KUKA KRL program: MyProgram_047().src

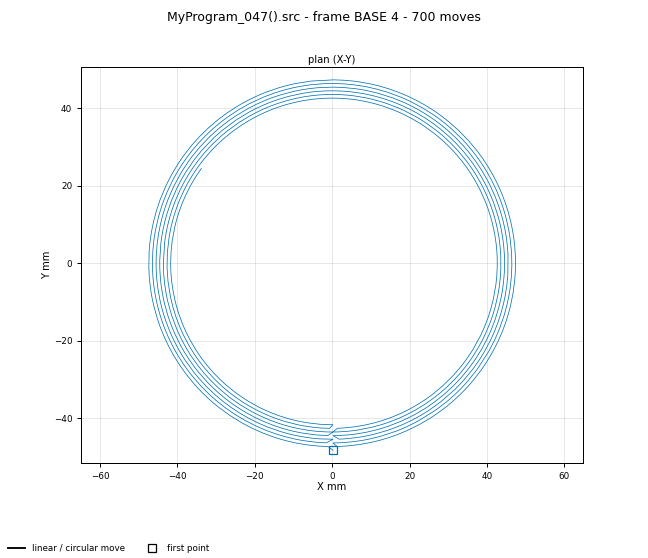
[picture p0: tool path of MyProgram_047().src in frame BASE 4, 700 of 700 moves have a stored position in this frame; points joined in program order, loops and branches not executed]
&ACCESS RVP
&REL 1
&PARAM TEMPLATE = C:\KRC\Roboter\Template\vorgabe
&PARAM EDITMASK = *
DEF MyProgram_047()
; ---- Setting reference (Base) ----
$BASE = BASE_DATA[4]

; --------------------------
; ---- Setting tool (TCP) ----
$TOOL = TOOL_DATA[3]
; --------------------------

$VEL.CP = VEL_APROX_PRINT
Startdeposition()
$VEL.CP = VEL_PRINT
LIN {X 0.2248,Y -48.3264,Z 65,A -97.1945,B 24.8798,C -2.5309,E1 24.997,E2 -179.1657} C_DIS
Enddeposition()
LIN {X 0.2248,Y -48.3264,Z 65,A -97.1945,B 24.8798,C -2.5309,E1 24.997,E2 -179.1657} C_DIS
Startdeposition()
$VEL.CP = VEL_PRINT
LIN {X -1.0477,Y -47.3732,Z 65,A -98.6326,B 24.878,C -2.5491,E1 24.9931,E2 -177.7706} C_DIS
LIN {X -3.5749,Y -47.2498,Z 65,A -101.1612,B 24.8772,C -2.5575,E1 24.9861,E2 -175.2611} C_DIS
LIN {X -6.5546,Y -46.929,Z 65,A -105.0891,B 24.8776,C -2.5533,E1 24.9752,E2 -171.3204} C_DIS
LIN {X -9.2778,Y -46.468,Z 65,A -107.7216,B 24.8764,C -2.5655,E1 24.968,E2 -168.7143} C_DIS
LIN {X -11.575,Y -45.9489,Z 65,A -110.7748,B 24.8766,C -2.5637,E1 24.9597,E2 -165.6528} C_DIS
LIN {X -13.521,Y -45.4144,Z 65,A -113.2414,B 24.8766,C -2.5649,E1 24.9531,E2 -163.1849} C_DIS
LIN {X -15.4389,Y -44.7995,Z 65,A -115.7196,B 24.8764,C -2.5661,E1 24.9465,E2 -160.7051} C_DIS
LIN {X -17.756,Y -43.932,Z 65,A -119.0552,B 24.8766,C -2.5637,E1 24.9378,E2 -157.3566} C_DIS
LIN {X -20.3496,Y -42.7927,Z 65,A -122.8119,B 24.8767,C -2.5626,E1 24.9282,E2 -153.588} C_DIS
LIN {X -23.3064,Y -41.2571,Z 65,A -126.6828,B 24.876,C -2.5702,E1 24.9188,E2 -149.7241} C_DIS
LIN {X -26.4858,Y -39.2912,Z 65,A -131.3289,B 24.8755,C -2.5752,E1 24.9079,E2 -145.0751} C_DIS
LIN {X -29.4186,Y -37.1461,Z 65,A -135.0423,B 24.8738,C -2.5924,E1 24.8996,E2 -141.3894} C_DIS
LIN {X -30.8579,Y -35.9594,Z 65,A -137.3147,B 24.8734,C -2.5964,E1 24.8948,E2 -139.1176} C_DIS
LIN {X -32.1607,Y -34.7995,Z 65,A -139.563,B 24.8732,C -2.5985,E1 24.8901,E2 -136.8654} C_DIS
LIN {X -33.7294,Y -33.2807,Z 65,A -142.3681,B 24.8729,C -2.6017,E1 24.8846,E2 -134.056} C_DIS
LIN {X -35.5399,Y -31.34,Z 65,A -146.1751,B 24.873,C -2.6005,E1 24.8774,E2 -130.2292} C_DIS
LIN {X -37.5818,Y -28.8599,Z 65,A -149.5808,B 24.8715,C -2.616,E1 24.8716,E2 -126.8446} C_DIS
LIN {X -39.2128,Y -26.6015,Z 65,A -153.0058,B 24.8708,C -2.6235,E1 24.8661,E2 -123.4206} C_DIS
LIN {X -40.9588,Y -23.8267,Z 65,A -156.7428,B 24.8695,C -2.6367,E1 24.8607,E2 -119.696} C_DIS
LIN {X -42.1995,Y -21.5519,Z 65,A -160.1247,B 24.869,C -2.6418,E1 24.8563,E2 -116.3083} C_DIS
LIN {X -43.292,Y -19.2649,Z 65,A -163.5194,B 24.8685,C -2.646,E1 24.8523,E2 -112.905} C_DIS
LIN {X -44.419,Y -16.5014,Z 65,A -166.5245,B 24.8667,C -2.6641,E1 24.8493,E2 -109.9264} C_DIS
LIN {X -45.1483,Y -14.3836,Z 65,A -169.6546,B 24.8665,C -2.6665,E1 24.8466,E2 -106.7842} C_DIS
LIN {X -46.0448,Y -11.1877,Z 65,A -173.5161,B 24.8651,C -2.6804,E1 24.8438,E2 -102.9335} C_DIS
LIN {X -46.5143,Y -9.0394,Z 65,A -175.9159,B 24.8639,C -2.6918,E1 24.8425,E2 -100.5468} C_DIS
LIN {X -46.7881,Y -7.4983,Z 65,A -177.7088,B 24.8632,C -2.6989,E1 24.8416,E2 -98.7601} C_DIS
LIN {X -47.0559,Y -5.5702,Z 65,A 179.5109,B 24.863,C -2.7007,E1 24.8406,E2 -95.9675} C_DIS
LIN {X -47.2538,Y -3.5244,Z 65,A 177.0172,B 24.8622,C -2.7083,E1 24.8401,E2 -93.477} C_DIS
LIN {X -47.3725,Y -1.0864,Z 65,A 173.6451,B 24.8618,C -2.7122,E1 24.8398,E2 -90.094} C_DIS
LIN {X -47.2852,Y 3.0683,Z 65,A 169.3289,B 24.8593,C -2.737,E1 24.8402,E2 -85.8111} C_DIS
LIN {X -47.1535,Y 4.676,Z 65,A 167.3632,B 24.8587,C -2.743,E1 24.8407,E2 -83.8478} C_DIS
LIN {X -46.9842,Y 6.1456,Z 65,A 165.4093,B 24.8583,C -2.7465,E1 24.8414,E2 -81.8907} C_DIS
LIN {X -46.6648,Y 8.2283,Z 65,A 162.772,B 24.8576,C -2.7533,E1 24.8426,E2 -79.254} C_DIS
LIN {X -46.1094,Y 10.9184,Z 65,A 159.2452,B 24.8568,C -2.761,E1 24.8447,E2 -75.725} C_DIS
LIN {X -45.3809,Y 13.634,Z 65,A 155.7906,B 24.8558,C -2.7708,E1 24.8473,E2 -72.2736} C_DIS
LIN {X -44.4848,Y 16.3215,Z 65,A 152.1165,B 24.855,C -2.778,E1 24.8507,E2 -68.596} C_DIS
LIN {X -42.9085,Y 20.1037,Z 65,A 148.0403,B 24.8523,C -2.8039,E1 24.8552,E2 -64.5593} C_DIS
LIN {X -41.5375,Y 22.8004,Z 65,A 143.2509,B 24.8527,C -2.7999,E1 24.8615,E2 -59.7346} C_DIS
LIN {X -39.7956,Y 25.7219,Z 65,A 139.6863,B 24.8508,C -2.8183,E1 24.8667,E2 -56.196} C_DIS
LIN {X -38.3081,Y 27.8889,Z 65,A 136.4395,B 24.85,C -2.8259,E1 24.8719,E2 -52.9515} C_DIS
LIN {X -36.3484,Y 30.399,Z 65,A 132.1204,B 24.8496,C -2.8296,E1 24.8795,E2 -48.6212} C_DIS
LIN {X -34.1939,Y 32.8036,Z 65,A 128.7989,B 24.8477,C -2.8469,E1 24.8858,E2 -45.3263} C_DIS
LIN {X -31.929,Y 35.0116,Z 65,A 124.5127,B 24.8475,C -2.8495,E1 24.8945,E2 -41.0286} C_DIS
LIN {X -29.3388,Y 37.2091,Z 65,A 120.4495,B 24.8464,C -2.8589,E1 24.9032,E2 -36.9725} C_DIS
LIN {X -27.2469,Y 38.7679,Z 65,A 117.7102,B 24.8451,C -2.8709,E1 24.9094,E2 -34.2523} C_DIS
LIN {X -25.1174,Y 40.1796,Z 65,A 114.1999,B 24.8451,C -2.8708,E1 24.9177,E2 -30.7304} C_DIS
LIN {X -23.0226,Y 41.4156,Z 65,A 111.5759,B 24.8441,C -2.8803,E1 24.924,E2 -28.1213} C_DIS
LIN {X -21.3498,Y 42.3027,Z 65,A 108.9226,B 24.8443,C -2.8788,E1 24.9306,E2 -25.4573} C_DIS
LIN {X -18.8516,Y 43.4731,Z 65,A 105.8781,B 24.8433,C -2.8879,E1 24.9383,E2 -22.427} C_DIS
LIN {X -17.1589,Y 44.1688,Z 65,A 103.2338,B 24.8437,C -2.8846,E1 24.9452,E2 -19.7692} C_DIS
LIN {X -13.7455,Y 45.3477,Z 65,A 99.3402,B 24.8424,C -2.8965,E1 24.9555,E2 -15.897} C_DIS
LIN {X -11.6308,Y 45.9347,Z 65,A 96.6918,B 24.8421,C -2.8993,E1 24.9626,E2 -13.2511} C_DIS
LIN {X -9.6114,Y 46.3995,Z 65,A 93.6894,B 24.8426,C -2.894,E1 24.9709,E2 -10.2324} C_DIS
LIN {X -5.4319,Y 47.0721,Z 65,A 87.9261,B 24.8433,C -2.8875,E1 24.9869,E2 -4.4493} C_DIS
LIN {X 0.4153,Y 47.3828,Z 65,A 82.2123,B 24.8408,C -2.9107,E1 25.0027,E2 1.2101} C_DIS
LIN {X 2.9923,Y 47.2903,Z 65,A 78.3924,B 24.842,C -2.8997,E1 25.0134,E2 5.0549} C_DIS
LIN {X 5.4396,Y 47.0712,Z 65,A 76.0531,B 24.8409,C -2.9094,E1 25.0198,E2 7.3696} C_DIS
LIN {X 6.891,Y 46.8812,Z 65,A 73.417,B 24.8425,C -2.8951,E1 25.0272,E2 10.0375} C_DIS
LIN {X 10.45,Y 46.2182,Z 65,A 69.7173,B 24.8415,C -2.9041,E1 25.0372,E2 13.7111} C_DIS
LIN {X 12.4414,Y 45.722,Z 65,A 67.3234,B 24.8415,C -2.9041,E1 25.0437,E2 16.1014} C_DIS
LIN {X 14.7365,Y 45.0349,Z 65,A 64.0648,B 24.8424,C -2.8959,E1 25.0524,E2 19.3735} C_DIS
LIN {X 17.1608,Y 44.1681,Z 65,A 61.5002,B 24.8417,C -2.9023,E1 25.0591,E2 21.9175} C_DIS
LIN {X 19.5293,Y 43.1728,Z 65,A 58.0138,B 24.8428,C -2.8925,E1 25.0681,E2 25.4187} C_DIS
LIN {X 22.0777,Y 41.9268,Z 65,A 54.4054,B 24.8436,C -2.8852,E1 25.0771,E2 29.0346} C_DIS
LIN {X 24.0287,Y 40.8401,Z 65,A 52.0557,B 24.8433,C -2.8875,E1 25.0827,E2 31.3718} C_DIS
LIN {X 26.0373,Y 39.5897,Z 65,A 49.0436,B 24.8441,C -2.8805,E1 25.0898,E2 34.3908} C_DIS
LIN {X 27.6805,Y 38.4592,Z 65,A 46.9948,B 24.8438,C -2.8829,E1 25.0945,E2 36.4268} C_DIS
LIN {X 30.0285,Y 36.6556,Z 65,A 42.6889,B 24.8459,C -2.8637,E1 25.104,E2 40.7623} C_DIS
LIN {X 32.6756,Y 34.3172,Z 65,A 39.2026,B 24.8453,C -2.8693,E1 25.1111,E2 44.2211} C_DIS
LIN {X 35.1657,Y 31.76,Z 65,A 33.5783,B 24.8488,C -2.8365,E1 25.122,E2 49.8986} C_DIS
LIN {X 37.3052,Y 29.2173,Z 65,A 30.3479,B 24.8483,C -2.8414,E1 25.1276,E2 53.1024} C_DIS
LIN {X 38.9389,Y 27.0008,Z 65,A 27.2515,B 24.8487,C -2.8376,E1 25.1326,E2 56.1928} C_DIS
LIN {X 40.0929,Y 25.2561,Z 65,A 24.5767,B 24.8497,C -2.8285,E1 25.1366,E2 58.8757} C_DIS
LIN {X 41.5557,Y 22.769,Z 65,A 21.3683,B 24.8501,C -2.8245,E1 25.141,E2 62.0768} C_DIS
LIN {X 42.6058,Y 20.7386,Z 65,A 18.7825,B 24.8506,C -2.8203,E1 25.1443,E2 64.6587} C_DIS
LIN {X 43.2405,Y 19.3793,Z 65,A 16.9517,B 24.8511,C -2.815,E1 25.1464,E2 66.4923} C_DIS
LIN {X 43.9147,Y 17.7984,Z 65,A 14.7277,B 24.8521,C -2.8064,E1 25.1488,E2 68.7244} C_DIS
LIN {X 44.6883,Y 15.7559,Z 65,A 11.9805,B 24.8531,C -2.7968,E1 25.1514,E2 71.479} C_DIS
LIN {X 45.5346,Y 13.1116,Z 65,A 8.6685,B 24.854,C -2.7877,E1 25.1541,E2 74.7935} C_DIS
LIN {X 46.1594,Y 10.7047,Z 65,A 5.7168,B 24.8549,C -2.7798,E1 25.1561,E2 77.747} C_DIS
LIN {X 46.6091,Y 8.5383,Z 65,A 3.2753,B 24.8552,C -2.7761,E1 25.1574,E2 80.183} C_DIS
LIN {X 46.9274,Y 6.5651,Z 65,A 0.7893,B 24.8562,C -2.7673,E1 25.1585,E2 82.675} C_DIS
LIN {X 47.1911,Y 4.2771,Z 65,A -2.3414,B 24.8577,C -2.7521,E1 25.1594,E2 85.8233} C_DIS
LIN {X 47.348,Y 1.8664,Z 65,A -5.3383,B 24.8588,C -2.7415,E1 25.1597,E2 88.8274} C_DIS
LIN {X 47.3497,Y -1.8254,Z 65,A -9.1955,B 24.8591,C -2.7391,E1 25.1597,E2 92.6674} C_DIS
LIN {X 47.2256,Y -3.8774,Z 65,A -12.3248,B 24.8612,C -2.7189,E1 25.1589,E2 95.8258} C_DIS
LIN {X 46.7501,Y -7.728,Z 65,A -16.4295,B 24.8615,C -2.7154,E1 25.1574,E2 99.9146} C_DIS
LIN {X 46.0614,Y -11.1191,Z 65,A -20.4864,B 24.8626,C -2.7048,E1 25.155,E2 103.9729} C_DIS
LIN {X 45.5564,Y -13.0349,Z 65,A -22.9569,B 24.8635,C -2.696,E1 25.1532,E2 106.4501} C_DIS
LIN {X 44.855,Y -15.2752,Z 65,A -25.9707,B 24.8647,C -2.6839,E1 25.1506,E2 109.4753} C_DIS
LIN {X 43.9991,Y -17.5908,Z 65,A -28.8384,B 24.8654,C -2.6772,E1 25.1477,E2 112.343} C_DIS
LIN {X 42.9253,Y -20.0675,Z 65,A -32.2517,B 24.8667,C -2.6647,E1 25.1438,E2 115.7674} C_DIS
LIN {X 41.3563,Y -23.1288,Z 65,A -36.8186,B 24.8686,C -2.6451,E1 25.1377,E2 120.3567} C_DIS
LIN {X 39.6698,Y -25.9158,Z 65,A -40.056,B 24.8684,C -2.6473,E1 25.1329,E2 123.5725} C_DIS
LIN {X 38.5931,Y -27.492,Z 65,A -42.6591,B 24.8696,C -2.6355,E1 25.1287,E2 126.1907} C_DIS
LIN {X 36.6666,Y -30.0149,Z 65,A -46.2346,B 24.8701,C -2.6304,E1 25.1226,E2 129.7615} C_DIS
LIN {X 35.1534,Y -31.7722,Z 65,A -49.1478,B 24.871,C -2.6214,E1 25.1172,E2 132.683} C_DIS
LIN {X 33.2247,Y -33.7848,Z 65,A -52.4808,B 24.8717,C -2.614,E1 25.1106,E2 136.0192} C_DIS
LIN {X 31.1855,Y -35.6756,Z 65,A -55.7244,B 24.8722,C -2.6085,E1 25.1039,E2 139.2628} C_DIS
LIN {X 29.4222,Y -37.1432,Z 65,A -58.7213,B 24.8732,C -2.5985,E1 25.0974,E2 142.2722} C_DIS
LIN {X 26.8221,Y -39.0614,Z 65,A -62.1627,B 24.8732,C -2.5991,E1 25.0896,E2 145.7001} C_DIS
LIN {X 25.2556,Y -40.0932,Z 65,A -64.5338,B 24.8738,C -2.5929,E1 25.084,E2 148.0781} C_DIS
LIN {X 22.4419,Y -41.7329,Z 65,A -69.0409,B 24.8754,C -2.5759,E1 25.073,E2 152.6122} C_DIS
LIN {X 19.3312,Y -43.2621,Z 65,A -72.9814,B 24.8756,C -2.5739,E1 25.0631,E2 156.5474} C_DIS
LIN {X 16.8162,Y -44.3001,Z 65,A -76.0254,B 24.8756,C -2.5736,E1 25.0552,E2 159.5852} C_DIS
LIN {X 14.54,Y -45.0985,Z 65,A -78.9796,B 24.8761,C -2.5694,E1 25.0473,E2 162.5436} C_DIS
LIN {X 12.2916,Y -45.7625,Z 65,A -81.7852,B 24.8763,C -2.5669,E1 25.0398,E2 165.3506} C_DIS
LIN {X 10.1313,Y -46.2887,Z 65,A -84.5563,B 24.8767,C -2.563,E1 25.0322,E2 168.1271} C_DIS
LIN {X 7.0707,Y -46.8542,Z 65,A -88.5388,B 24.8773,C -2.5565,E1 25.0212,E2 172.1209} C_DIS
LIN {X 3.8207,Y -47.2301,Z 65,A -92.1846,B 24.877,C -2.5595,E1 25.0111,E2 175.7572} C_DIS
LIN {X 1.2789,Y -47.3675,Z 65,A -95.8986,B 24.8781,C -2.5481,E1 25.0007,E2 179.4974} C_DIS
LIN {X 1.2789,Y -47.3675,Z 65,A -95.8986,B 24.8781,C -2.5481,E1 25.0007,E2 179.4974} C_DIS
Enddeposition()
LIN {X 0.234,Y -46.4396,Z 65,A -96.8007,B 24.876,C -2.5704,E1 24.9983,E2 180.3466} C_DIS
Startdeposition()
$VEL.CP = VEL_PRINT
LIN {X 2.4648,Y -46.3766,Z 65,A -92.4422,B 24.8734,C -2.5972,E1 25.0107,E2 175.9252} C_DIS
LIN {X 5.2271,Y -46.1472,Z 65,A -88.7775,B 24.8728,C -2.6031,E1 25.0209,E2 172.2488} C_DIS
LIN {X 7.9459,Y -45.7575,Z 65,A -85.477,B 24.8727,C -2.604,E1 25.03,E2 168.9492} C_DIS
LIN {X 10.1123,Y -45.3281,Z 65,A -83.0608,B 24.873,C -2.6012,E1 25.0366,E2 166.543} C_DIS
LIN {X 12.7412,Y -44.6601,Z 65,A -78.8302,B 24.8711,C -2.6199,E1 25.0481,E2 162.2746} C_DIS
LIN {X 16.6628,Y -43.3497,Z 65,A -74.2326,B 24.8714,C -2.6176,E1 25.0601,E2 157.692} C_DIS
LIN {X 19.0595,Y -42.3508,Z 65,A -71.362,B 24.8714,C -2.6164,E1 25.0674,E2 154.8311} C_DIS
LIN {X 22.1501,Y -40.8195,Z 65,A -66.0149,B 24.8688,C -2.643,E1 25.0808,E2 149.4359} C_DIS
LIN {X 26.9328,Y -37.8344,Z 65,A -59.4392,B 24.8682,C -2.6494,E1 25.0961,E2 142.8669} C_DIS
LIN {X 30.0243,Y -35.431,Z 65,A -54.8607,B 24.8676,C -2.6551,E1 25.106,E2 138.2921} C_DIS
LIN {X 31.9687,Y -33.6883,Z 65,A -52.268,B 24.868,C -2.6509,E1 25.1112,E2 135.7199} C_DIS
LIN {X 33.1131,Y -32.5636,Z 65,A -50.4093,B 24.8678,C -2.6534,E1 25.1149,E2 133.8633} C_DIS
LIN {X 34.9088,Y -30.6307,Z 65,A -46.5756,B 24.8659,C -2.6722,E1 25.1221,E2 130.0019} C_DIS
LIN {X 37.4038,Y -27.5273,Z 65,A -41.0638,B 24.8634,C -2.6965,E1 25.1316,E2 124.4588} C_DIS
LIN {X 40.4448,Y -22.8258,Z 65,A -34.4215,B 24.862,C -2.7107,E1 25.1412,E2 117.8168} C_DIS
LIN {X 42.0103,Y -19.7997,Z 65,A -30.9945,B 24.8623,C -2.7081,E1 25.1454,E2 114.4144} C_DIS
LIN {X 43.0408,Y -17.4457,Z 65,A -27.3594,B 24.8604,C -2.7264,E1 25.1493,E2 110.7558} C_DIS
LIN {X 44.4285,Y -13.5269,Z 65,A -22.3166,B 24.859,C -2.7404,E1 25.1538,E2 105.7084} C_DIS
LIN {X 45.1092,Y -11.0463,Z 65,A -19.7706,B 24.8592,C -2.7382,E1 25.1555,E2 103.1823} C_DIS
LIN {X 45.5719,Y -8.9492,Z 65,A -16.8117,B 24.8577,C -2.7524,E1 25.1572,E2 100.2071} C_DIS
LIN {X 45.9664,Y -6.63,Z 65,A -14.0872,B 24.8571,C -2.7581,E1 25.1584,E2 97.4852} C_DIS
LIN {X 46.3142,Y -3.4512,Z 65,A -10.412,B 24.8564,C -2.7653,E1 25.1594,E2 93.8147} C_DIS
LIN {X 46.4375,Y -0.6361,Z 65,A -6.2616,B 24.8539,C -2.7892,E1 25.1598,E2 89.6324} C_DIS
LIN {X 46.363,Y 2.7109,Z 65,A -1.9539,B 24.8521,C -2.8056,E1 25.1592,E2 85.3116} C_DIS
LIN {X 45.93,Y 6.8774,Z 65,A 2.6288,B 24.8516,C -2.8102,E1 25.1577,E2 80.7449} C_DIS
LIN {X 45.6088,Y 8.7574,Z 65,A 5.6403,B 24.8495,C -2.8301,E1 25.1561,E2 77.7041} C_DIS
LIN {X 44.7769,Y 12.3244,Z 65,A 9.3288,B 24.8498,C -2.8277,E1 25.1536,E2 74.0425} C_DIS
LIN {X 44.2174,Y 14.2015,Z 65,A 11.6057,B 24.8493,C -2.8321,E1 25.1517,E2 71.768} C_DIS
LIN {X 43.4228,Y 16.4715,Z 65,A 15.0599,B 24.8474,C -2.8499,E1 25.1484,E2 68.2911} C_DIS
LIN {X 42.5233,Y 18.6718,Z 65,A 18.1112,B 24.8463,C -2.8604,E1 25.145,E2 65.2318} C_DIS
LIN {X 41.2763,Y 21.2873,Z 65,A 21.0738,B 24.8465,C -2.8586,E1 25.1413,E2 62.2892} C_DIS
LIN {X 40.0787,Y 23.4634,Z 65,A 24.8095,B 24.8442,C -2.8792,E1 25.1361,E2 58.5241} C_DIS
LIN {X 38.746,Y 25.6048,Z 65,A 27.6638,B 24.8439,C -2.8822,E1 25.1318,E2 55.6768} C_DIS
LIN {X 36.8655,Y 28.2454,Z 65,A 31.2343,B 24.8437,C -2.8839,E1 25.1259,E2 52.1195} C_DIS
LIN {X 34.8813,Y 30.6622,Z 65,A 35.0703,B 24.8428,C -2.8923,E1 25.119,E2 48.2811} C_DIS
LIN {X 33.5459,Y 32.1178,Z 65,A 38.0555,B 24.8412,C -2.9075,E1 25.1132,E2 45.273} C_DIS
LIN {X 30.5761,Y 34.9565,Z 65,A 42.4025,B 24.8415,C -2.9046,E1 25.1044,E2 40.9506} C_DIS
LIN {X 29.3534,Y 35.9896,Z 65,A 44.4539,B 24.8409,C -2.9096,E1 25.0999,E2 38.8951} C_DIS
LIN {X 27.9127,Y 37.1179,Z 65,A 46.6995,B 24.8405,C -2.9133,E1 25.095,E2 36.6488} C_DIS
LIN {X 26.4482,Y 38.1753,Z 65,A 49.416,B 24.8392,C -2.9256,E1 25.0887,E2 33.9127} C_DIS
LIN {X 23.3065,Y 40.1709,Z 65,A 54.1731,B 24.8381,C -2.9351,E1 25.0773,E2 29.1478} C_DIS
LIN {X 19.9982,Y 41.9156,Z 65,A 58.174,B 24.8386,C -2.9303,E1 25.0674,E2 25.1693} C_DIS
LIN {X 17.8551,Y 42.8729,Z 65,A 61.4383,B 24.8376,C -2.9396,E1 25.059,E2 21.8906} C_DIS
LIN {X 14.4147,Y 44.1484,Z 65,A 66.116,B 24.8369,C -2.946,E1 25.0467,E2 17.2071} C_DIS
LIN {X 11.7257,Y 44.9376,Z 65,A 69.1464,B 24.8374,C -2.9411,E1 25.0386,E2 14.1932} C_DIS
LIN {X 9.0679,Y 45.5489,Z 65,A 72.403,B 24.8374,C -2.9409,E1 25.0297,E2 10.9412} C_DIS
LIN {X 7.1132,Y 45.894,Z 65,A 74.8567,B 24.8374,C -2.9418,E1 25.0229,E2 8.488} C_DIS
LIN {X 4.9617,Y 46.1763,Z 65,A 77.5049,B 24.8374,C -2.9418,E1 25.0156,E2 5.8418} C_DIS
LIN {X 2.938,Y 46.3493,Z 65,A 80.0529,B 24.8373,C -2.9426,E1 25.0085,E2 3.2931} C_DIS
LIN {X 1.0284,Y 46.4309,Z 65,A 82.2696,B 24.8376,C -2.9402,E1 25.0023,E2 1.0827} C_DIS
LIN {X -2.0746,Y 46.3957,Z 65,A 87.1042,B 24.8359,C -2.9548,E1 24.9887,E2 -3.7874} C_DIS
LIN {X -5.6226,Y 46.1009,Z 65,A 90.6473,B 24.8376,C -2.9394,E1 24.979,E2 -7.2959} C_DIS
LIN {X -8.0541,Y 45.7385,Z 65,A 93.8831,B 24.8376,C -2.9404,E1 24.9701,E2 -10.5369} C_DIS
LIN {X -10.1044,Y 45.3299,Z 65,A 96.0806,B 24.8384,C -2.9325,E1 24.9641,E2 -12.7183} C_DIS
LIN {X -12.24,Y 44.8001,Z 65,A 99.1519,B 24.8381,C -2.9351,E1 24.9558,E2 -15.8004} C_DIS
LIN {X -14.9072,Y 43.9845,Z 65,A 102.735,B 24.8383,C -2.9333,E1 24.9462,E2 -19.3856} C_DIS
LIN {X -17.556,Y 42.9958,Z 65,A 106.411,B 24.8385,C -2.9314,E1 24.9367,E2 -23.065} C_DIS
LIN {X -21.3543,Y 41.2421,Z 65,A 110.9502,B 24.8404,C -2.9145,E1 24.9253,E2 -27.5757} C_DIS
LIN {X -24.0772,Y 39.7133,Z 65,A 115.5671,B 24.8399,C -2.9186,E1 24.9141,E2 -32.2161} C_DIS
LIN {X -26.977,Y 37.8034,Z 65,A 119.584,B 24.8413,C -2.9066,E1 24.9049,E2 -36.2178} C_DIS
LIN {X -29.0485,Y 36.2367,Z 65,A 122.508,B 24.8424,C -2.896,E1 24.8985,E2 -39.1274} C_DIS
LIN {X -30.8599,Y 34.7066,Z 65,A 125.6094,B 24.8429,C -2.892,E1 24.892,E2 -42.2312} C_DIS
LIN {X -32.6866,Y 32.9916,Z 65,A 128.6329,B 24.8437,C -2.8839,E1 24.8859,E2 -45.248} C_DIS
LIN {X -34.4284,Y 31.1706,Z 65,A 131.8654,B 24.8444,C -2.878,E1 24.8798,E2 -48.4806} C_DIS
LIN {X -36.0562,Y 29.2712,Z 65,A 134.897,B 24.8453,C -2.8695,E1 24.8744,E2 -51.5058} C_DIS
LIN {X -37.3433,Y 27.6112,Z 65,A 137.2919,B 24.8463,C -2.8601,E1 24.8703,E2 -53.8896} C_DIS
LIN {X -38.7934,Y 25.5329,Z 65,A 140.9211,B 24.8465,C -2.8582,E1 24.8646,E2 -57.5325} C_DIS
LIN {X -40.1542,Y 23.3355,Z 65,A 143.7107,B 24.848,C -2.8441,E1 24.8607,E2 -60.3027} C_DIS
LIN {X -41.1959,Y 21.4416,Z 65,A 146.861,B 24.8482,C -2.8428,E1 24.8565,E2 -63.4664} C_DIS
LIN {X -42.6418,Y 18.3987,Z 65,A 150.6903,B 24.8499,C -2.8263,E1 24.8521,E2 -67.2773} C_DIS
LIN {X -43.5502,Y 16.1335,Z 65,A 153.613,B 24.851,C -2.8161,E1 24.8492,E2 -70.1922} C_DIS
LIN {X -44.1917,Y 14.2811,Z 65,A 156.1423,B 24.8516,C -2.8102,E1 24.847,E2 -72.7218} C_DIS
LIN {X -44.8242,Y 12.151,Z 65,A 159.2751,B 24.852,C -2.8068,E1 24.8446,E2 -75.8645} C_DIS
LIN {X -45.6661,Y 8.4571,Z 65,A 163.6858,B 24.8539,C -2.7889,E1 24.8421,E2 -80.2583} C_DIS
LIN {X -46.0564,Y 5.9714,Z 65,A 166.7164,B 24.855,C -2.7782,E1 24.8409,E2 -83.2815} C_DIS
LIN {X -46.3058,Y 3.5563,Z 65,A 169.8512,B 24.8558,C -2.7706,E1 24.8401,E2 -86.4169} C_DIS
LIN {X -46.437,Y 0.6959,Z 65,A 173.5953,B 24.8567,C -2.7622,E1 24.8398,E2 -90.1634} C_DIS
LIN {X -46.399,Y -1.9968,Z 65,A 176.7575,B 24.858,C -2.7497,E1 24.84,E2 -93.3148} C_DIS
LIN {X -46.2717,Y -3.9822,Z 65,A 178.8665,B 24.8592,C -2.7377,E1 24.8405,E2 -95.4078} C_DIS
LIN {X -46.0878,Y -5.7275,Z 65,A -178.7723,B 24.8597,C -2.7335,E1 24.8412,E2 -97.773} C_DIS
LIN {X -45.8261,Y -7.5393,Z 65,A -176.5889,B 24.8605,C -2.7256,E1 24.8422,E2 -99.9506} C_DIS
LIN {X -45.4232,Y -9.6765,Z 65,A -173.6984,B 24.861,C -2.7201,E1 24.8438,E2 -102.8451} C_DIS
LIN {X -44.8712,Y -11.9767,Z 65,A -170.8524,B 24.862,C -2.7105,E1 24.8457,E2 -105.6845} C_DIS
LIN {X -44.1446,Y -14.4257,Z 65,A -167.621,B 24.8629,C -2.7023,E1 24.8484,E2 -108.9149} C_DIS
LIN {X -43.3813,Y -16.5813,Z 65,A -164.723,B 24.8636,C -2.6952,E1 24.8512,E2 -111.8123} C_DIS
LIN {X -42.3444,Y -19.0737,Z 65,A -161.8833,B 24.8652,C -2.6794,E1 24.8543,E2 -114.6301} C_DIS
LIN {X -41.2849,Y -21.2689,Z 65,A -158.0636,B 24.8649,C -2.682,E1 24.859,E2 -118.4765} C_DIS
LIN {X -39.9763,Y -23.6378,Z 65,A -154.9009,B 24.866,C -2.6709,E1 24.8634,E2 -121.6291} C_DIS
LIN {X -38.5305,Y -25.9283,Z 65,A -151.8991,B 24.8673,C -2.6579,E1 24.8679,E2 -124.6151} C_DIS
LIN {X -37.6446,Y -27.1995,Z 65,A -149.9162,B 24.8677,C -2.6542,E1 24.8712,E2 -126.5989} C_DIS
LIN {X -36.3842,Y -28.8626,Z 65,A -146.8875,B 24.8677,C -2.6544,E1 24.8764,E2 -129.6423} C_DIS
LIN {X -33.9635,Y -31.6761,Z 65,A -142.0783,B 24.8684,C -2.6476,E1 24.8853,E2 -134.4567} C_DIS
LIN {X -31.4889,Y -34.1367,Z 65,A -138.1278,B 24.8697,C -2.6339,E1 24.8933,E2 -138.3908} C_DIS
LIN {X -29.5934,Y -35.7924,Z 65,A -135.1317,B 24.8705,C -2.6266,E1 24.8996,E2 -141.3811} C_DIS
LIN {X -27.5671,Y -37.375,Z 65,A -131.5769,B 24.8705,C -2.6266,E1 24.9076,E2 -144.9488} C_DIS
LIN {X -25.2527,Y -38.9759,Z 65,A -128.2622,B 24.8712,C -2.6189,E1 24.9153,E2 -148.2561} C_DIS
LIN {X -22.6134,Y -40.5646,Z 65,A -124.8035,B 24.8722,C -2.6086,E1 24.9236,E2 -151.7007} C_DIS
LIN {X -19.5151,Y -42.1429,Z 65,A -120.3621,B 24.8725,C -2.6057,E1 24.9347,E2 -156.1469} C_DIS
LIN {X -17.0667,Y -43.1925,Z 65,A -116.8053,B 24.8725,C -2.6066,E1 24.9439,E2 -159.7136} C_DIS
LIN {X -14.6993,Y -44.0546,Z 65,A -113.6668,B 24.8726,C -2.6045,E1 24.9522,E2 -162.8533} C_DIS
LIN {X -12.1101,Y -44.8353,Z 65,A -109.9662,B 24.8723,C -2.6081,E1 24.9622,E2 -166.5682} C_DIS
LIN {X -9.1432,Y -45.5335,Z 65,A -106.9243,B 24.8736,C -2.5951,E1 24.9704,E2 -169.583} C_DIS
LIN {X -7.4996,Y -45.8326,Z 65,A -104.4536,B 24.873,C -2.601,E1 24.9772,E2 -172.0701} C_DIS
LIN {X -4.1492,Y -46.2564,Z 65,A -100.8544,B 24.8739,C -2.5914,E1 24.9872,E2 -175.6487} C_DIS
LIN {X -1.4825,Y -46.4183,Z 65,A -96.8776,B 24.8728,C -2.6027,E1 24.9983,E2 -179.6534} C_DIS
LIN {X -1.4825,Y -46.4183,Z 65,A -96.8776,B 24.8728,C -2.6027,E1 24.9983,E2 -179.6534} C_DIS
Enddeposition()
LIN {X 0.224,Y -45.4804,Z 65,A -95.5777,B 24.8724,C -2.6065,E1 25.002,E2 -180.9623} C_DIS
Startdeposition()
$VEL.CP = VEL_PRINT
LIN {X -3.2271,Y -45.3852,Z 65,A -100.777,B 24.8738,C -2.5924,E1 24.9874,E2 -175.7285} C_DIS
LIN {X -5.068,Y -45.2164,Z 65,A -103.0617,B 24.8738,C -2.5932,E1 24.981,E2 -173.4445} C_DIS
LIN {X -6.6649,Y -45.0091,Z 65,A -105.2906,B 24.874,C -2.5906,E1 24.9749,E2 -171.2076} C_DIS
LIN {X -9.0087,Y -44.5989,Z 65,A -108.3653,B 24.874,C -2.5905,E1 24.9664,E2 -168.1294} C_DIS
LIN {X -11.1576,Y -44.1105,Z 65,A -110.8903,B 24.8735,C -2.5956,E1 24.9596,E2 -165.6132} C_DIS
LIN {X -13.3396,Y -43.5002,Z 65,A -114.1911,B 24.874,C -2.591,E1 24.9507,E2 -162.2958} C_DIS
LIN {X -16.8989,Y -42.2446,Z 65,A -119.0434,B 24.8737,C -2.5938,E1 24.938,E2 -157.4401} C_DIS
LIN {X -19.1263,Y -41.2842,Z 65,A -121.4828,B 24.8725,C -2.6058,E1 24.9318,E2 -155.0235} C_DIS
LIN {X -21.3788,Y -40.1645,Z 65,A -124.5738,B 24.872,C -2.6107,E1 24.9241,E2 -151.9361} C_DIS
LIN {X -23.7976,Y -38.7802,Z 65,A -128.7004,B 24.8724,C -2.607,E1 24.9141,E2 -147.7881} C_DIS
LIN {X -25.9506,Y -37.3734,Z 65,A -131.8407,B 24.8718,C -2.6135,E1 24.9069,E2 -144.6527} C_DIS
LIN {X -28.0665,Y -35.8121,Z 65,A -135.1269,B 24.8712,C -2.6195,E1 24.8996,E2 -141.3691} C_DIS
LIN {X -30.1938,Y -34.0371,Z 65,A -138.3281,B 24.8701,C -2.6299,E1 24.8928,E2 -138.1802} C_DIS
LIN {X -32.4723,Y -31.8711,Z 65,A -142.4448,B 24.8695,C -2.6358,E1 24.8846,E2 -134.0605} C_DIS
LIN {X -34.3409,Y -29.848,Z 65,A -145.9488,B 24.8688,C -2.6429,E1 24.878,E2 -130.5579} C_DIS
LIN {X -35.7092,Y -28.1967,Z 65,A -149.0971,B 24.8688,C -2.6434,E1 24.8725,E2 -127.3959} C_DIS
LIN {X -37.8475,Y -25.2546,Z 65,A -153.2379,B 24.8671,C -2.6602,E1 24.8659,E2 -123.275} C_DIS
LIN {X -38.9924,Y -23.4486,Z 65,A -155.8262,B 24.8663,C -2.6684,E1 24.8621,E2 -120.693} C_DIS
LIN {X -39.7714,Y -22.1008,Z 65,A -158.1071,B 24.8662,C -2.6695,E1 24.8589,E2 -118.4028} C_DIS
LIN {X -41.0557,Y -19.611,Z 65,A -161.4057,B 24.8649,C -2.6819,E1 24.8548,E2 -115.1163} C_DIS
LIN {X -41.8318,Y -17.8988,Z 65,A -164.3154,B 24.8649,C -2.6818,E1 24.8516,E2 -112.1901} C_DIS
LIN {X -42.9197,Y -15.1032,Z 65,A -167.6519,B 24.8633,C -2.698,E1 24.8483,E2 -108.8737} C_DIS
LIN {X -43.5436,Y -13.1994,Z 65,A -170.2099,B 24.8626,C -2.705,E1 24.8462,E2 -106.3176} C_DIS
LIN {X -44.0964,Y -11.2124,Z 65,A -172.6652,B 24.8616,C -2.7145,E1 24.8444,E2 -103.8707} C_DIS
LIN {X -44.4878,Y -9.5427,Z 65,A -174.9494,B 24.8611,C -2.7194,E1 24.843,E2 -101.585} C_DIS
LIN {X -45.0187,Y -6.5999,Z 65,A -178.6815,B 24.8599,C -2.7313,E1 24.8413,E2 -97.8592} C_DIS
LIN {X -45.3058,Y -4.1938,Z 65,A 178.2738,B 24.8589,C -2.7409,E1 24.8403,E2 -94.8191} C_DIS
LIN {X -45.4346,Y -2.4291,Z 65,A 176.0299,B 24.8582,C -2.7476,E1 24.8399,E2 -92.5779} C_DIS
LIN {X -45.4935,Y -0.7413,Z 65,A 173.6894,B 24.8578,C -2.7517,E1 24.8398,E2 -90.233} C_DIS
LIN {X -45.4745,Y 1.5114,Z 65,A 170.4521,B 24.8574,C -2.7558,E1 24.84,E2 -86.9861} C_DIS
LIN {X -45.2191,Y 5.0456,Z 65,A 166.2831,B 24.8555,C -2.7733,E1 24.841,E2 -82.834} C_DIS
LIN {X -44.852,Y 7.65,Z 65,A 163.2479,B 24.8541,C -2.787,E1 24.8423,E2 -79.8135} C_DIS
LIN {X -44.3258,Y 10.2676,Z 65,A 159.2462,B 24.8538,C -2.7898,E1 24.8446,E2 -75.7948} C_DIS
LIN {X -43.6869,Y 12.7164,Z 65,A 156.5695,B 24.8521,C -2.8057,E1 24.8466,E2 -73.1407} C_DIS
LIN {X -43.0662,Y 14.6808,Z 65,A 153.6741,B 24.8517,C -2.81,E1 24.8491,E2 -70.2389} C_DIS
LIN {X -42.3612,Y 16.6051,Z 65,A 150.0279,B 24.8522,C -2.805,E1 24.8529,E2 -66.5603} C_DIS
LIN {X -40.9853,Y 19.7589,Z 65,A 146.2193,B 24.8502,C -2.8239,E1 24.8574,E2 -62.7762} C_DIS
LIN {X -38.9452,Y 23.5263,Z 65,A 140.8096,B 24.8486,C -2.839,E1 24.8649,E2 -57.3743} C_DIS
LIN {X -37.2173,Y 26.1745,Z 65,A 137.3271,B 24.8468,C -2.8559,E1 24.8703,E2 -53.915} C_DIS
LIN {X -36.1488,Y 27.6315,Z 65,A 135.2552,B 24.8458,C -2.8644,E1 24.8738,E2 -51.8534} C_DIS
LIN {X -34.1734,Y 30.0388,Z 65,A 130.6967,B 24.8456,C -2.8663,E1 24.882,E2 -47.2787} C_DIS
LIN {X -31.6247,Y 32.7116,Z 65,A 125.9166,B 24.8446,C -2.8757,E1 24.8914,E2 -42.5007} C_DIS
LIN {X -29.2062,Y 34.8888,Z 65,A 122.4832,B 24.8427,C -2.8932,E1 24.8986,E2 -39.0957} C_DIS
LIN {X -26.8754,Y 36.7139,Z 65,A 118.0301,B 24.8429,C -2.8914,E1 24.9085,E2 -34.6224} C_DIS
LIN {X -24.9566,Y 38.0445,Z 65,A 115.1401,B 24.8422,C -2.8976,E1 24.9153,E2 -31.7376} C_DIS
LIN {X -21.5508,Y 40.0723,Z 65,A 110.656,B 24.8405,C -2.913,E1 24.9261,E2 -27.2771} C_DIS
LIN {X -19.5683,Y 41.0763,Z 65,A 107.8011,B 24.8402,C -2.9166,E1 24.9332,E2 -24.4232} C_DIS
LIN {X -17.3621,Y 42.0572,Z 65,A 104.8929,B 24.8395,C -2.9227,E1 24.9407,E2 -21.5229} C_DIS
LIN {X -15.6037,Y 42.7402,Z 65,A 102.3552,B 24.8394,C -2.9235,E1 24.9473,E2 -18.9818} C_DIS
LIN {X -13.3623,Y 43.4933,Z 65,A 99.0942,B 24.8394,C -2.923,E1 24.956,E2 -15.7137} C_DIS
LIN {X -9.9326,Y 44.4023,Z 65,A 95.186,B 24.8381,C -2.9352,E1 24.9665,E2 -11.8289} C_DIS
LIN {X -7.7712,Y 44.8305,Z 65,A 92.3016,B 24.8381,C -2.9357,E1 24.9744,E2 -8.9427} C_DIS
LIN {X -5.8139,Y 45.1265,Z 65,A 89.7638,B 24.8379,C -2.9366,E1 24.9815,E2 -6.4051} C_DIS
LIN {X -3.8125,Y 45.3393,Z 65,A 86.5819,B 24.8389,C -2.9284,E1 24.9904,E2 -3.202} C_DIS
LIN {X 0.06,Y 45.5,Z 65,A 82.147,B 24.838,C -2.9363,E1 25.0027,E2 1.2146} C_DIS
LIN {X 2.7755,Y 45.4155,Z 65,A 78.3746,B 24.8386,C -2.9311,E1 25.0132,E2 4.998} C_DIS
LIN {X 5.9384,Y 45.1104,Z 65,A 75.1318,B 24.8373,C -2.9422,E1 25.0222,E2 8.2124} C_DIS
LIN {X 7.336,Y 44.9041,Z 65,A 73.2338,B 24.8376,C -2.9398,E1 25.0274,E2 10.1141} C_DIS
LIN {X 8.9306,Y 44.615,Z 65,A 70.8461,B 24.8383,C -2.9335,E1 25.034,E2 12.5139} C_DIS
LIN {X 11.8092,Y 43.9403,Z 65,A 66.6447,B 24.8394,C -2.9239,E1 25.0454,E2 16.7318} C_DIS
LIN {X 15.6838,Y 42.711,Z 65,A 62.2024,B 24.8386,C -2.9305,E1 25.0571,E2 21.1498} C_DIS
LIN {X 18.603,Y 41.5227,Z 65,A 58.4473,B 24.8386,C -2.9299,E1 25.0667,E2 24.8976} C_DIS
LIN {X 20.5752,Y 40.5818,Z 65,A 55.2724,B 24.8398,C -2.9196,E1 25.0747,E2 28.0884} C_DIS
LIN {X 22.6379,Y 39.468,Z 65,A 52.8828,B 24.8392,C -2.925,E1 25.0805,E2 30.4583} C_DIS
LIN {X 24.543,Y 38.3125,Z 65,A 49.5531,B 24.8407,C -2.912,E1 25.0885,E2 33.8082} C_DIS
LIN {X 26.6412,Y 36.8848,Z 65,A 46.5273,B 24.8409,C -2.9096,E1 25.0954,E2 36.8292} C_DIS
LIN {X 28.1443,Y 35.7506,Z 65,A 44.4522,B 24.8409,C -2.9105,E1 25.0999,E2 38.8946} C_DIS
LIN {X 29.7834,Y 34.3975,Z 65,A 41.2761,B 24.8423,C -2.8969,E1 25.1068,E2 42.0906} C_DIS
LIN {X 31.8511,Y 32.4921,Z 65,A 37.4633,B 24.8436,C -2.8851,E1 25.1145,E2 45.9157} C_DIS
LIN {X 33.8887,Y 30.3604,Z 65,A 34.444,B 24.8432,C -2.8891,E1 25.1202,E2 48.9122} C_DIS
LIN {X 35.3861,Y 28.6011,Z 65,A 31.3251,B 24.8443,C -2.8788,E1 25.1257,E2 52.0413} C_DIS
LIN {X 37.1367,Y 26.2886,Z 65,A 27.4182,B 24.8457,C -2.8655,E1 25.1322,E2 55.9608} C_DIS
LIN {X 38.5479,Y 24.1716,Z 65,A 24.2587,B 24.8465,C -2.8582,E1 25.137,E2 59.1218} C_DIS
LIN {X 40.1581,Y 21.3902,Z 65,A 20.8241,B 24.8465,C -2.8585,E1 25.1416,E2 62.5378} C_DIS
LIN {X 40.8075,Y 20.1236,Z 65,A 18.2428,B 24.8485,C -2.8394,E1 25.1449,E2 65.1504} C_DIS
LIN {X 42.2125,Y 16.9802,Z 65,A 14.2921,B 24.8491,C -2.8342,E1 25.1492,E2 69.0919} C_DIS
LIN {X 43.1991,Y 14.2867,Z 65,A 11.0666,B 24.8495,C -2.8307,E1 25.1522,E2 72.3074} C_DIS
LIN {X 43.7467,Y 12.5072,Z 65,A 8.7483,B 24.8501,C -2.8243,E1 25.154,E2 74.6276} C_DIS
LIN {X 44.1683,Y 10.9263,Z 65,A 6.6306,B 24.8509,C -2.8171,E1 25.1555,E2 76.7502} C_DIS
LIN {X 44.6052,Y 8.9772,Z 65,A 4.0813,B 24.8518,C -2.8089,E1 25.157,E2 79.3041} C_DIS
LIN {X 44.9625,Y 6.9694,Z 65,A 1.582,B 24.8525,C -2.8023,E1 25.1581,E2 81.8044} C_DIS
LIN {X 45.2406,Y 4.8481,Z 65,A -1.3082,B 24.8537,C -2.7903,E1 25.1591,E2 84.7058} C_DIS
LIN {X 45.4427,Y 2.283,Z 65,A -5.2844,B 24.8562,C -2.7667,E1 25.1597,E2 88.7143} C_DIS
LIN {X 45.3988,Y -3.0258,Z 65,A -10.738,B 24.856,C -2.7684,E1 25.1594,E2 94.1313} C_DIS
LIN {X 45.1331,Y -5.7633,Z 65,A -14.8743,B 24.8585,C -2.7451,E1 25.1581,E2 98.2984} C_DIS
LIN {X 44.7124,Y -8.4278,Z 65,A -17.8498,B 24.8588,C -2.7422,E1 25.1567,E2 101.2633} C_DIS
LIN {X 44.257,Y -10.5626,Z 65,A -20.5581,B 24.8596,C -2.7344,E1 25.155,E2 103.9743} C_DIS
LIN {X 43.5288,Y -13.2452,Z 65,A -24.5883,B 24.8617,C -2.7139,E1 25.1519,E2 108.0299} C_DIS
LIN {X 42.7503,Y -15.576,Z 65,A -27.4256,B 24.8622,C -2.7092,E1 25.1492,E2 110.8624} C_DIS
LIN {X 41.7901,Y -17.9952,Z 65,A -30.431,B 24.8626,C -2.7044,E1 25.146,E2 113.8626} C_DIS
LIN {X 40.833,Y -20.0721,Z 65,A -33.5707,B 24.864,C -2.6912,E1 25.1422,E2 117.0166} C_DIS
LIN {X 39.3465,Y -22.8494,Z 65,A -37.1441,B 24.8644,C -2.687,E1 25.1374,E2 120.5812} C_DIS
LIN {X 38.2722,Y -24.6057,Z 65,A -39.7432,B 24.8652,C -2.6797,E1 25.1335,E2 123.1845} C_DIS
LIN {X 36.4353,Y -27.2521,Z 65,A -44.2601,B 24.8671,C -2.6605,E1 25.1262,E2 127.7249} C_DIS
LIN {X 33.8822,Y -30.3668,Z 65,A -49.8079,B 24.8692,C -2.6393,E1 25.116,E2 133.2979} C_DIS
LIN {X 31.7066,Y -32.6332,Z 65,A -53.7496,B 24.8701,C -2.6302,E1 25.1082,E2 137.2447} C_DIS
LIN {X 28.0891,Y -35.7942,Z 65,A -59.2872,B 24.8705,C -2.6259,E1 25.0963,E2 142.7711} C_DIS
LIN {X 24.8341,Y -38.1249,Z 65,A -63.8204,B 24.8706,C -2.6248,E1 25.0859,E2 147.2914} C_DIS
LIN {X 22.9134,Y -39.309,Z 65,A -66.6784,B 24.8712,C -2.6193,E1 25.079,E2 150.1534} C_DIS
LIN {X 20.7131,Y -40.5114,Z 65,A -70.0922,B 24.8721,C -2.6097,E1 25.0706,E2 153.5805} C_DIS
LIN {X 18.2848,Y -41.6639,Z 65,A -73.1244,B 24.8721,C -2.6105,E1 25.0629,E2 156.6031} C_DIS
LIN {X 16.4339,Y -42.4283,Z 65,A -76.0941,B 24.8731,C -2.5996,E1 25.0552,E2 159.5921} C_DIS
LIN {X 14.2165,Y -43.2218,Z 65,A -79.1708,B 24.8737,C -2.5941,E1 25.047,E2 162.6758} C_DIS
LIN {X 10.7189,Y -44.2189,Z 65,A -83.246,B 24.8733,C -2.5977,E1 25.036,E2 166.7361} C_DIS
LIN {X 8.3913,Y -44.7186,Z 65,A -86.1114,B 24.8733,C -2.5973,E1 25.0282,E2 169.5989} C_DIS
LIN {X 6.5346,Y -45.028,Z 65,A -88.8842,B 24.8741,C -2.5892,E1 25.0205,E2 172.3885} C_DIS
LIN {X 3.1933,Y -45.3871,Z 65,A -92.5138,B 24.8734,C -2.5965,E1 25.0105,E2 175.9983} C_DIS
LIN {X 1.806,Y -45.4638,Z 65,A -95.5063,B 24.8754,C -2.5765,E1 25.002,E2 179.0377} C_DIS
LIN {X 1.806,Y -45.4638,Z 65,A -95.5063,B 24.8754,C -2.5765,E1 25.002,E2 179.0377} C_DIS
Enddeposition()
LIN {X 0.2255,Y -44.5448,Z 65,A -96.2858,B 24.872,C -2.6115,E1 25.0001,E2 179.734} C_DIS
Startdeposition()
$VEL.CP = VEL_PRINT
LIN {X 1.4173,Y -44.5345,Z 65,A -93.5709,B 24.8701,C -2.6302,E1 25.0077,E2 176.9751} C_DIS
LIN {X 4.2396,Y -44.3549,Z 65,A -90.1004,B 24.8702,C -2.6292,E1 25.0174,E2 173.5086} C_DIS
LIN {X 6.3435,Y -44.1032,Z 65,A -87.307,B 24.8699,C -2.6321,E1 25.0251,E2 170.7108} C_DIS
LIN {X 9.1021,Y -43.6174,Z 65,A -83.5243,B 24.8693,C -2.6379,E1 25.0355,E2 166.9185} C_DIS
LIN {X 11.9017,Y -42.9381,Z 65,A -79.7582,B 24.8689,C -2.6427,E1 25.0457,E2 163.1469} C_DIS
LIN {X 14.5786,Y -42.1049,Z 65,A -75.9718,B 24.8681,C -2.6501,E1 25.0558,E2 159.3503} C_DIS
LIN {X 18.2287,Y -40.6577,Z 65,A -71.5984,B 24.8686,C -2.6458,E1 25.067,E2 154.9971} C_DIS
LIN {X 21.2746,Y -39.15,Z 65,A -66.3493,B 24.8663,C -2.6681,E1 25.0801,E2 149.7098} C_DIS
LIN {X 24.1257,Y -37.4604,Z 65,A -62.7961,B 24.8668,C -2.6636,E1 25.0885,E2 146.1785} C_DIS
LIN {X 26.2977,Y -35.9689,Z 65,A -59.2802,B 24.8659,C -2.6726,E1 25.0965,E2 142.6535} C_DIS
LIN {X 28.8516,Y -33.9546,Z 65,A -54.6786,B 24.8642,C -2.6891,E1 25.1065,E2 138.0303} C_DIS
LIN {X 31.2004,Y -31.8102,Z 65,A -51.2089,B 24.8644,C -2.6875,E1 25.1135,E2 134.5787} C_DIS
LIN {X 33.4032,Y -29.4883,Z 65,A -46.636,B 24.8625,C -2.7059,E1 25.1222,E2 129.9824} C_DIS
LIN {X 35.4997,Y -26.9278,Z 65,A -42.6309,B 24.8618,C -2.7124,E1 25.1291,E2 125.9806} C_DIS
LIN {X 37.0184,Y -24.7992,Z 65,A -39.5875,B 24.8615,C -2.7157,E1 25.1339,E2 122.9444} C_DIS
LIN {X 38.6888,Y -22.1024,Z 65,A -34.7151,B 24.8588,C -2.7418,E1 25.1409,E2 118.0353} C_DIS
LIN {X 40.1077,Y -19.4091,Z 65,A -31.8418,B 24.8596,C -2.7339,E1 25.1445,E2 115.1958} C_DIS
LIN {X 41.1696,Y -17.0419,Z 65,A -27.8695,B 24.8574,C -2.7556,E1 25.1489,E2 111.1941} C_DIS
LIN {X 42.1875,Y -14.3362,Z 65,A -24.2896,B 24.8565,C -2.7643,E1 25.1522,E2 107.6137} C_DIS
LIN {X 43.0739,Y -11.4024,Z 65,A -20.5003,B 24.8555,C -2.7736,E1 25.1551,E2 103.824} C_DIS
LIN {X 43.7202,Y -8.594,Z 65,A -17.2942,B 24.8553,C -2.7759,E1 25.157,E2 100.6311} C_DIS
LIN {X 43.9571,Y -7.2871,Z 65,A -15.2661,B 24.8541,C -2.7872,E1 25.158,E2 98.5882} C_DIS
LIN {X 44.2935,Y -4.8405,Z 65,A -12.0536,B 24.853,C -2.7979,E1 25.1591,E2 95.3695} C_DIS
LIN {X 44.4995,Y -2.2526,Z 65,A -8.1216,B 24.8507,C -2.8194,E1 25.1597,E2 91.4098} C_DIS
LIN {X 44.5074,Y 2.1112,Z 65,A -3.2826,B 24.8503,C -2.8226,E1 25.1595,E2 86.5921} C_DIS
LIN {X 44.3341,Y 4.4554,Z 65,A -0.4424,B 24.8497,C -2.8286,E1 25.1588,E2 83.7544} C_DIS
LIN {X 44.0682,Y 6.5853,Z 65,A 2.6141,B 24.8482,C -2.8426,E1 25.1577,E2 80.6829} C_DIS
LIN {X 43.7374,Y 8.5071,Z 65,A 4.7408,B 24.8482,C -2.8433,E1 25.1566,E2 78.5671} C_DIS
LIN {X 43.4124,Y 10.0344,Z 65,A 6.7161,B 24.8475,C -2.8487,E1 25.1554,E2 76.5903} C_DIS
LIN {X 42.8862,Y 12.0872,Z 65,A 10.0102,B 24.8455,C -2.8673,E1 25.153,E2 73.2713} C_DIS
LIN {X 41.7227,Y 15.6386,Z 65,A 14.8378,B 24.844,C -2.8816,E1 25.1485,E2 68.437} C_DIS
LIN {X 40.8211,Y 17.8596,Z 65,A 17.2709,B 24.8443,C -2.8784,E1 25.1459,E2 66.0246} C_DIS
LIN {X 39.9081,Y 19.816,Z 65,A 20.1922,B 24.8432,C -2.8887,E1 25.1424,E2 63.0948} C_DIS
LIN {X 38.9035,Y 21.7219,Z 65,A 23.041,B 24.8423,C -2.8975,E1 25.1386,E2 60.2401} C_DIS
LIN {X 37.5961,Y 23.9143,Z 65,A 26.1675,B 24.8416,C -2.9031,E1 25.134,E2 57.1162} C_DIS
LIN {X 36.3026,Y 25.835,Z 65,A 29.3707,B 24.8404,C -2.9144,E1 25.1289,E2 53.9019} C_DIS
LIN {X 35.0764,Y 27.4768,Z 65,A 31.706,B 24.8403,C -2.9154,E1 25.1249,E2 51.5754} C_DIS
LIN {X 34.1287,Y 28.6462,Z 65,A 33.9882,B 24.8391,C -2.9259,E1 25.1208,E2 49.2788} C_DIS
LIN {X 32.2725,Y 30.7227,Z 65,A 37.627,B 24.8382,C -2.9347,E1 25.1139,E2 45.6352} C_DIS
LIN {X 30.3874,Y 32.5878,Z 65,A 41.199,B 24.8371,C -2.9444,E1 25.1067,E2 42.055} C_DIS
LIN {X 28.0032,Y 34.6576,Z 65,A 44.6896,B 24.8373,C -2.9422,E1 25.0993,E2 38.5831} C_DIS
LIN {X 26.1232,Y 36.0959,Z 65,A 47.927,B 24.8364,C -2.9507,E1 25.092,E2 35.3371} C_DIS
LIN {X 24.0618,Y 37.5014,Z 65,A 51.1395,B 24.8358,C -2.9557,E1 25.0845,E2 32.1231} C_DIS
LIN {X 21.9413,Y 38.7808,Z 65,A 54.1321,B 24.8357,C -2.957,E1 25.0773,E2 29.1366} C_DIS
LIN {X 20.223,Y 39.7029,Z 65,A 57.1228,B 24.8344,C -2.9682,E1 25.0699,E2 26.1277} C_DIS
LIN {X 18.1399,Y 40.6977,Z 65,A 59.7874,B 24.8346,C -2.9665,E1 25.0631,E2 23.4738} C_DIS
LIN {X 15.8972,Y 41.6248,Z 65,A 62.7043,B 24.8346,C -2.9663,E1 25.0556,E2 20.5639} C_DIS
LIN {X 13.6198,Y 42.4245,Z 65,A 66.1139,B 24.8338,C -2.9737,E1 25.0465,E2 17.1433} C_DIS
LIN {X 11.0289,Y 43.1705,Z 65,A 69.3548,B 24.834,C -2.9723,E1 25.0378,E2 13.9109} C_DIS
LIN {X 8.7933,Y 43.681,Z 65,A 72.3634,B 24.8337,C -2.9746,E1 25.0296,E2 10.9008} C_DIS
LIN {X 6.6624,Y 44.0563,Z 65,A 74.9224,B 24.834,C -2.9721,E1 25.0225,E2 8.3504} C_DIS
LIN {X 4.9033,Y 44.2868,Z 65,A 77.3002,B 24.8338,C -2.9739,E1 25.0159,E2 5.9699} C_DIS
LIN {X 3.0927,Y 44.4496,Z 65,A 79.5593,B 24.8338,C -2.9729,E1 25.0097,E2 3.7145} C_DIS
LIN {X 0.9408,Y 44.5472,Z 65,A 82.4136,B 24.8338,C -2.9739,E1 25.0017,E2 0.8585} C_DIS
LIN {X -1.5404,Y 44.5307,Z 65,A 85.8934,B 24.8334,C -2.9774,E1 24.992,E2 -2.63} C_DIS
LIN {X -3.7596,Y 44.3986,Z 65,A 88.3423,B 24.8342,C -2.9701,E1 24.9852,E2 -5.0626} C_DIS
LIN {X -5.3116,Y 44.2394,Z 65,A 90.2432,B 24.8345,C -2.9675,E1 24.9799,E2 -6.9584} C_DIS
LIN {X -7.3681,Y 43.9436,Z 65,A 93.5161,B 24.8337,C -2.9744,E1 24.9708,E2 -10.2507} C_DIS
LIN {X -11.2554,Y 43.1119,Z 65,A 98.8608,B 24.8339,C -2.9731,E1 24.9563,E2 -15.5994} C_DIS
LIN {X -13.9718,Y 42.3104,Z 65,A 101.8735,B 24.8353,C -2.9602,E1 24.9483,E2 -18.5865} C_DIS
LIN {X -15.9507,Y 41.6045,Z 65,A 104.8067,B 24.8353,C -2.9599,E1 24.9407,E2 -21.5252} C_DIS
LIN {X -17.868,Y 40.8175,Z 65,A 107.328,B 24.836,C -2.9542,E1 24.9342,E2 -24.0388} C_DIS
LIN {X -19.7414,Y 39.945,Z 65,A 110.2447,B 24.836,C -2.9537,E1 24.9269,E2 -26.9616} C_DIS
LIN {X -21.4555,Y 39.0518,Z 65,A 113.2244,B 24.8358,C -2.9562,E1 24.9195,E2 -29.9558} C_DIS
LIN {X -24.5716,Y 37.1694,Z 65,A 117.8846,B 24.8368,C -2.9472,E1 24.9086,E2 -34.6096} C_DIS
LIN {X -28.4379,Y 34.3018,Z 65,A 122.8084,B 24.84,C -2.9179,E1 24.8978,E2 -39.4811} C_DIS
LIN {X -30.5076,Y 32.4748,Z 65,A 127.7865,B 24.8389,C -2.9283,E1 24.8874,E2 -44.5042} C_DIS
LIN {X -33.7685,Y 29.07,Z 65,A 133.9241,B 24.8404,C -2.9144,E1 24.8759,E2 -50.6357} C_DIS
LIN {X -35.6293,Y 26.7559,Z 65,A 137.5825,B 24.8417,C -2.9024,E1 24.8697,E2 -54.2828} C_DIS
LIN {X -37.8647,Y 23.4864,Z 65,A 142.0225,B 24.8441,C -2.8803,E1 24.8629,E2 -58.6923} C_DIS
LIN {X -39.1478,Y 21.2786,Z 65,A 145.7994,B 24.8445,C -2.8771,E1 24.8578,E2 -62.4814} C_DIS
LIN {X -40.213,Y 19.19,Z 65,A 148.9132,B 24.8453,C -2.8695,E1 24.854,E2 -65.5939} C_DIS
LIN {X -41.588,Y 15.9938,Z 65,A 153.1054,B 24.8471,C -2.8527,E1 24.8496,E2 -69.7693} C_DIS
LIN {X -42.7065,Y 12.7076,Z 65,A 157.3087,B 24.8489,C -2.836,E1 24.846,E2 -73.9566} C_DIS
LIN {X -43.2639,Y 10.6567,Z 65,A 160.1788,B 24.8496,C -2.8292,E1 24.844,E2 -76.8273} C_DIS
LIN {X -43.6591,Y 8.9,Z 65,A 162.2153,B 24.8507,C -2.8187,E1 24.8428,E2 -78.8505} C_DIS
LIN {X -44.0149,Y 6.9303,Z 65,A 164.9787,B 24.8514,C -2.8129,E1 24.8415,E2 -81.6164} C_DIS
LIN {X -44.2489,Y 5.2309,Z 65,A 168.0167,B 24.851,C -2.8161,E1 24.8405,E2 -84.6802} C_DIS
LIN {X -44.5513,Y 0.7177,Z 65,A 173.2622,B 24.8537,C -2.7908,E1 24.8398,E2 -89.8969} C_DIS
LIN {X -44.5303,Y -1.537,Z 65,A 176.3322,B 24.8544,C -2.7838,E1 24.84,E2 -92.9687} C_DIS
LIN {X -44.3393,Y -4.4055,Z 65,A 179.6868,B 24.8561,C -2.7682,E1 24.8407,E2 -96.306} C_DIS
LIN {X -44.1251,Y -6.189,Z 65,A -178.0442,B 24.8569,C -2.7606,E1 24.8416,E2 -98.5703} C_DIS
LIN {X -43.6717,Y -8.8387,Z 65,A -174.6913,B 24.8581,C -2.7488,E1 24.8432,E2 -101.9148} C_DIS
LIN {X -43.3162,Y -10.4426,Z 65,A -171.9842,B 24.858,C -2.7497,E1 24.8449,E2 -104.64} C_DIS
LIN {X -42.4855,Y -13.4284,Z 65,A -168.3045,B 24.8596,C -2.7342,E1 24.8478,E2 -108.3039} C_DIS
LIN {X -41.5974,Y -15.9695,Z 65,A -164.2936,B 24.8599,C -2.7311,E1 24.8517,E2 -112.33} C_DIS
LIN {X -40.7335,Y -18.0605,Z 65,A -161.1256,B 24.8604,C -2.7262,E1 24.8553,E2 -115.5038} C_DIS
LIN {X -39.0746,Y -21.4134,Z 65,A -157.0193,B 24.8626,C -2.7044,E1 24.8605,E2 -119.5799} C_DIS
LIN {X -38.0049,Y -23.2587,Z 65,A -154.4502,B 24.8636,C -2.6951,E1 24.8642,E2 -122.1401} C_DIS
LIN {X -37.1638,Y -24.5801,Z 65,A -152.0451,B 24.8636,C -2.6951,E1 24.8679,E2 -124.557} C_DIS
LIN {X -35.4148,Y -27.0397,Z 65,A -148.5752,B 24.8651,C -2.6804,E1 24.8735,E2 -128.0089} C_DIS
LIN {X -34.5752,Y -28.1048,Z 65,A -145.4487,B 24.8636,C -2.6945,E1 24.8792,E2 -131.1836} C_DIS
LIN {X -31.9689,Y -31.0377,Z 65,A -141.2268,B 24.8659,C -2.6727,E1 24.8871,E2 -135.3719} C_DIS
LIN {X -29.8602,Y -33.0716,Z 65,A -137.2892,B 24.8664,C -2.6676,E1 24.8952,E2 -139.3132} C_DIS
LIN {X -27.39,Y -35.1448,Z 65,A -133.5892,B 24.8677,C -2.654,E1 24.9032,E2 -142.9948} C_DIS
LIN {X -25.7509,Y -36.3626,Z 65,A -131.0504,B 24.8683,C -2.6485,E1 24.9089,E2 -145.5293} C_DIS
LIN {X -24.4217,Y -37.2682,Z 65,A -128.7501,B 24.8683,C -2.6485,E1 24.9143,E2 -147.8371} C_DIS
LIN {X -22.2941,Y -38.5779,Z 65,A -125.5378,B 24.8687,C -2.6439,E1 24.922,E2 -151.0484} C_DIS
LIN {X -20.0367,Y -39.7977,Z 65,A -122.1408,B 24.869,C -2.6411,E1 24.9304,E2 -154.4481} C_DIS
LIN {X -17.8056,Y -40.8446,Z 65,A -118.9546,B 24.8693,C -2.638,E1 24.9385,E2 -157.6345} C_DIS
LIN {X -15.1834,Y -41.8903,Z 65,A -115.44,B 24.8698,C -2.633,E1 24.9476,E2 -161.1446} C_DIS
LIN {X -12.964,Y -42.63,Z 65,A -112.3907,B 24.87,C -2.6313,E1 24.9558,E2 -164.1955} C_DIS
LIN {X -11.1696,Y -43.1343,Z 65,A -110.279,B 24.8705,C -2.6257,E1 24.9614,E2 -166.297} C_DIS
LIN {X -9.6375,Y -43.5025,Z 65,A -108.2014,B 24.8705,C -2.6255,E1 24.9671,E2 -168.3768} C_DIS
LIN {X -7.5668,Y -43.9098,Z 65,A -105.0438,B 24.87,C -2.6313,E1 24.9758,E2 -171.5514} C_DIS
LIN {X -4.2182,Y -44.3564,Z 65,A -100.9277,B 24.8704,C -2.6272,E1 24.9872,E2 -175.6605} C_DIS
LIN {X -1.138,Y -44.5425,Z 65,A -96.3467,B 24.8694,C -2.6371,E1 25,E2 -180.266} C_DIS
LIN {X -1.138,Y -44.5425,Z 65,A -96.3467,B 24.8694,C -2.6371,E1 25,E2 -180.266} C_DIS
Enddeposition()
LIN {X 0.2144,Y -43.6138,Z 65,A -95.5656,B 24.8693,C -2.6387,E1 25.0022,E2 -181.0508} C_DIS
Startdeposition()
$VEL.CP = VEL_PRINT
LIN {X -1.3845,Y -43.5926,Z 65,A -99.0035,B 24.8713,C -2.6182,E1 24.9925,E2 -177.5641} C_DIS
LIN {X -3.8619,Y -43.4433,Z 65,A -102.0192,B 24.8709,C -2.6218,E1 24.9841,E2 -174.5557} C_DIS
LIN {X -6.1538,Y -43.1782,Z 65,A -105.1312,B 24.8709,C -2.6212,E1 24.9755,E2 -171.44} C_DIS
LIN {X -8.7396,Y -42.7299,Z 65,A -108.4161,B 24.8706,C -2.6247,E1 24.9665,E2 -168.1601} C_DIS
LIN {X -10.7013,Y -42.281,Z 65,A -111.0595,B 24.8706,C -2.6261,E1 24.9593,E2 -165.5162} C_DIS
LIN {X -12.5676,Y -41.7649,Z 65,A -113.5451,B 24.8703,C -2.6286,E1 24.9526,E2 -163.0325} C_DIS
LIN {X -14.4024,Y -41.1679,Z 65,A -116.2287,B 24.8703,C -2.6285,E1 24.9455,E2 -160.3437} C_DIS
LIN {X -16.283,Y -40.4613,Z 65,A -118.7333,B 24.8698,C -2.6328,E1 24.939,E2 -157.844} C_DIS
LIN {X -18.5785,Y -39.4596,Z 65,A -122.8153,B 24.8705,C -2.6257,E1 24.9286,E2 -153.7351} C_DIS
LIN {X -20.7383,Y -38.3686,Z 65,A -125.8937,B 24.87,C -2.6311,E1 24.921,E2 -150.6609} C_DIS
LIN {X -23.7353,Y -36.591,Z 65,A -129.9311,B 24.8686,C -2.6448,E1 24.9115,E2 -146.6437} C_DIS
LIN {X -25.5504,Y -35.3479,Z 65,A -132.6913,B 24.868,C -2.6512,E1 24.9052,E2 -143.8892} C_DIS
LIN {X -26.713,Y -34.4769,Z 65,A -135.1119,B 24.8683,C -2.6479,E1 24.8998,E2 -141.4519} C_DIS
LIN {X -29.4319,Y -32.1868,Z 65,A -139.8611,B 24.8676,C -2.6558,E1 24.8898,E2 -136.7029} C_DIS
LIN {X -31.5802,Y -30.0829,Z 65,A -143.1983,B 24.866,C -2.6717,E1 24.8833,E2 -133.3893} C_DIS
LIN {X -33.1474,Y -28.3457,Z 65,A -146.7934,B 24.866,C -2.672,E1 24.8766,E2 -129.7789} C_DIS
LIN {X -34.8232,Y -26.2598,Z 65,A -150.6384,B 24.8655,C -2.6763,E1 24.87,E2 -125.9258} C_DIS
LIN {X -36.4798,Y -23.9053,Z 65,A -153.8072,B 24.8638,C -2.693,E1 24.8651,E2 -122.7812} C_DIS
LIN {X -37.7181,Y -21.9,Z 65,A -157.155,B 24.8633,C -2.6979,E1 24.8603,E2 -119.4281} C_DIS
LIN {X -38.89,Y -19.7436,Z 65,A -160.625,B 24.8627,C -2.7037,E1 24.8558,E2 -115.9533} C_DIS
LIN {X -40.034,Y -17.3067,Z 65,A -164.3512,B 24.8619,C -2.7113,E1 24.8516,E2 -112.2248} C_DIS
LIN {X -41.4681,Y -13.5142,Z 65,A -169.7664,B 24.8605,C -2.7257,E1 24.8466,E2 -106.8132} C_DIS
LIN {X -42.53,Y -9.667,Z 65,A -174.0898,B 24.8578,C -2.7519,E1 24.8436,E2 -102.5274} C_DIS
LIN {X -42.8067,Y -8.3561,Z 65,A -176.4712,B 24.8579,C -2.7501,E1 24.8423,E2 -100.1275} C_DIS
LIN {X -43.2846,Y -5.3598,Z 65,A 179.9608,B 24.8562,C -2.7671,E1 24.8408,E2 -96.5789} C_DIS
LIN {X -43.5325,Y -2.6806,Z 65,A 175.6085,B 24.856,C -2.7688,E1 24.8399,E2 -92.2047} C_DIS
LIN {X -43.6146,Y -0.0878,Z 65,A 171.688,B 24.8555,C -2.7738,E1 24.8399,E2 -88.2725} C_DIS
LIN {X -43.2773,Y 5.4166,Z 65,A 165.6563,B 24.8516,C -2.8102,E1 24.8412,E2 -82.2917} C_DIS
LIN {X -42.9872,Y 7.3709,Z 65,A 162.9269,B 24.8509,C -2.8168,E1 24.8424,E2 -79.5618} C_DIS
LIN {X -42.5616,Y 9.5266,Z 65,A 159.8073,B 24.8503,C -2.8231,E1 24.8442,E2 -76.4389} C_DIS
LIN {X -41.9561,Y 11.9126,Z 65,A 156.9038,B 24.8488,C -2.8368,E1 24.8463,E2 -73.5514} C_DIS
LIN {X -41.3164,Y 13.9706,Z 65,A 153.728,B 24.8483,C -2.8415,E1 24.849,E2 -70.3686} C_DIS
LIN {X -40.4956,Y 16.1971,Z 65,A 150.6189,B 24.8473,C -2.851,E1 24.8521,E2 -67.2646} C_DIS
LIN {X -39.332,Y 18.8472,Z 65,A 147.1386,B 24.8457,C -2.8658,E1 24.8561,E2 -63.8008} C_DIS
LIN {X -38.3495,Y 20.7736,Z 65,A 143.9413,B 24.8453,C -2.8699,E1 24.8603,E2 -60.5961} C_DIS
LIN {X -37.3174,Y 22.5754,Z 65,A 141.4583,B 24.8441,C -2.8804,E1 24.8638,E2 -58.1254} C_DIS
LIN {X -36.3021,Y 24.1747,Z 65,A 138.4998,B 24.844,C -2.8816,E1 24.8683,E2 -55.155} C_DIS
LIN {X -34.6907,Y 26.4355,Z 65,A 135.2749,B 24.8424,C -2.8963,E1 24.8736,E2 -51.9496} C_DIS
LIN {X -32.9501,Y 28.5752,Z 65,A 131.0113,B 24.8422,C -2.8978,E1 24.8813,E2 -47.67} C_DIS
LIN {X -31.0545,Y 30.6242,Z 65,A 127.6261,B 24.8409,C -2.91,E1 24.8878,E2 -44.2993} C_DIS
LIN {X -28.7413,Y 32.805,Z 65,A 123.4651,B 24.8398,C -2.9196,E1 24.8963,E2 -40.1445} C_DIS
LIN {X -27.1573,Y 34.1281,Z 65,A 120.1412,B 24.84,C -2.9179,E1 24.9036,E2 -36.804} C_DIS
LIN {X -24.0031,Y 36.4153,Z 65,A 115.6314,B 24.8381,C -2.9354,E1 24.9139,E2 -32.3207} C_DIS
LIN {X -21.4272,Y 37.9886,Z 65,A 111.9934,B 24.8368,C -2.9466,E1 24.9226,E2 -28.6983} C_DIS
LIN {X -19.7713,Y 38.8755,Z 65,A 109.3639,B 24.8366,C -2.9485,E1 24.9291,E2 -26.0662} C_DIS
LIN {X -18.0047,Y 39.7249,Z 65,A 106.6411,B 24.8364,C -2.9505,E1 24.936,E2 -23.3412} C_DIS
LIN {X -16.0746,Y 40.5444,Z 65,A 103.8986,B 24.836,C -2.9544,E1 24.9431,E2 -20.6019} C_DIS
LIN {X -14.0315,Y 41.2959,Z 65,A 101.0231,B 24.8356,C -2.9577,E1 24.9506,E2 -17.7287} C_DIS
LIN {X -11.6185,Y 42.0393,Z 65,A 97.4749,B 24.8356,C -2.9581,E1 24.9601,E2 -14.1757} C_DIS
LIN {X -9.2187,Y 42.6292,Z 65,A 94.585,B 24.8347,C -2.9659,E1 24.968,E2 -11.3004} C_DIS
LIN {X -7.2261,Y 43.0117,Z 65,A 91.821,B 24.8347,C -2.9665,E1 24.9756,E2 -8.5351} C_DIS
LIN {X -5.2397,Y 43.2989,Z 65,A 89.2529,B 24.8343,C -2.9691,E1 24.9827,E2 -5.9711} C_DIS
LIN {X -3.2624,Y 43.4928,Z 65,A 86.541,B 24.8343,C -2.9688,E1 24.9902,E2 -3.2574} C_DIS
LIN {X -1.2843,Y 43.5956,Z 65,A 83.9935,B 24.8342,C -2.9705,E1 24.9973,E2 -0.7132} C_DIS
LIN {X 0.466,Y 43.6125,Z 65,A 81.8212,B 24.8339,C -2.9727,E1 25.0034,E2 1.4536} C_DIS
LIN {X 2.278,Y 43.5552,Z 65,A 79.2907,B 24.8341,C -2.9707,E1 25.0104,E2 3.9882} C_DIS
LIN {X 4.15,Y 43.4168,Z 65,A 76.8368,B 24.8341,C -2.9707,E1 25.0173,E2 6.4407} C_DIS
LIN {X 5.6697,Y 43.2445,Z 65,A 74.1044,B 24.8354,C -2.9597,E1 25.0249,E2 9.1971} C_DIS
LIN {X 8.656,Y 42.7471,Z 65,A 70.9536,B 24.8342,C -2.9704,E1 25.0335,E2 12.3188} C_DIS
LIN {X 10.2426,Y 42.3948,Z 65,A 68.6311,B 24.8346,C -2.9665,E1 25.0398,E2 14.6475} C_DIS
LIN {X 12.4242,Y 41.8075,Z 65,A 65.7985,B 24.8346,C -2.9665,E1 25.0474,E2 17.4751} C_DIS
LIN {X 14.1934,Y 41.2407,Z 65,A 62.9962,B 24.8354,C -2.9591,E1 25.0548,E2 20.2899} C_DIS
LIN {X 17.1958,Y 40.0823,Z 65,A 59.2339,B 24.8351,C -2.9621,E1 25.0645,E2 24.0365} C_DIS
LIN {X 18.5426,Y 39.4768,Z 65,A 56.8025,B 24.8362,C -2.9522,E1 25.0707,E2 26.4852} C_DIS
LIN {X 21.2427,Y 38.0916,Z 65,A 53.3364,B 24.8359,C -2.9553,E1 25.0793,E2 29.9342} C_DIS
LIN {X 22.7241,Y 37.227,Z 65,A 50.9252,B 24.8365,C -2.9495,E1 25.0851,E2 32.3516} C_DIS
LIN {X 24.3976,Y 36.1523,Z 65,A 48.0429,B 24.8375,C -2.9411,E1 25.0918,E2 35.2443} C_DIS
LIN {X 26.9393,Y 34.3004,Z 65,A 44.5621,B 24.8371,C -2.9446,E1 25.0995,E2 38.7043} C_DIS
LIN {X 28.5228,Y 32.9953,Z 65,A 41.3887,B 24.8385,C -2.9317,E1 25.1064,E2 41.8961} C_DIS
LIN {X 30.3827,Y 31.2913,Z 65,A 37.9359,B 24.8395,C -2.9227,E1 25.1134,E2 45.356} C_DIS
LIN {X 32.5453,Y 29.0351,Z 65,A 33.6333,B 24.8408,C -2.9105,E1 25.1215,E2 49.6684} C_DIS
LIN {X 34.8358,Y 26.243,Z 65,A 29.389,B 24.8411,C -2.9079,E1 25.1289,E2 53.8991} C_DIS
LIN {X 36.1033,Y 24.4699,Z 65,A 26.7833,B 24.8414,C -2.9053,E1 25.133,E2 56.4982} C_DIS
LIN {X 36.9093,Y 23.2368,Z 65,A 24.5366,B 24.8425,C -2.895,E1 25.1364,E2 58.758} C_DIS
LIN {X 38.1327,Y 21.1681,Z 65,A 21.3585,B 24.8435,C -2.8864,E1 25.1409,E2 61.94} C_DIS
LIN {X 39.0086,Y 19.5084,Z 65,A 19.1922,B 24.8436,C -2.8849,E1 25.1436,E2 64.0983} C_DIS
LIN {X 39.911,Y 17.5888,Z 65,A 16.2071,B 24.8448,C -2.8738,E1 25.1471,E2 67.0938} C_DIS
LIN {X 40.8274,Y 15.3415,Z 65,A 12.896,B 24.846,C -2.8625,E1 25.1505,E2 70.413} C_DIS
LIN {X 41.6936,Y 12.8016,Z 65,A 9.5738,B 24.8468,C -2.8558,E1 25.1533,E2 73.7323} C_DIS
LIN {X 42.2928,Y 10.6579,Z 65,A 6.5496,B 24.8479,C -2.8453,E1 25.1555,E2 76.7639} C_DIS
LIN {X 42.7699,Y 8.5442,Z 65,A 3.9835,B 24.8483,C -2.8417,E1 25.157,E2 79.3238} C_DIS
LIN {X 43.0978,Y 6.694,Z 65,A 1.3464,B 24.8494,C -2.8311,E1 25.1582,E2 81.9703} C_DIS
LIN {X 43.3943,Y 4.3759,Z 65,A -1.7998,B 24.8506,C -2.8203,E1 25.1592,E2 85.1236} C_DIS
LIN {X 43.5714,Y 1.9393,Z 65,A -5.1878,B 24.852,C -2.8071,E1 25.1597,E2 88.5227} C_DIS
LIN {X 43.5899,Y -1.4705,Z 65,A -9.0349,B 24.8523,C -2.8043,E1 25.1597,E2 92.3535} C_DIS
LIN {X 43.48,Y -3.4233,Z 65,A -11.935,B 24.8538,C -2.7903,E1 25.1591,E2 95.2695} C_DIS
LIN {X 43.2132,Y -5.9063,Z 65,A -15.184,B 24.8548,C -2.7805,E1 25.158,E2 98.5223} C_DIS
LIN {X 42.9232,Y -7.7344,Z 65,A -18.0178,B 24.8563,C -2.7658,E1 25.1566,E2 101.3745} C_DIS
LIN {X 42.148,Y -11.2162,Z 65,A -22.2227,B 24.8569,C -2.7598,E1 25.1539,E2 105.5692} C_DIS
LIN {X 41.4537,Y -13.5587,Z 65,A -25.2301,B 24.8576,C -2.7535,E1 25.1514,E2 108.5742} C_DIS
LIN {X 40.8809,Y -15.2,Z 65,A -27.8106,B 24.8589,C -2.7414,E1 25.1489,E2 111.1691} C_DIS
LIN {X 39.6376,Y -18.1972,Z 65,A -31.801,B 24.8597,C -2.7335,E1 25.1445,E2 115.1563} C_DIS
LIN {X 38.725,Y -20.065,Z 65,A -34.4399,B 24.8603,C -2.7272,E1 25.1412,E2 117.796} C_DIS
LIN {X 37.594,Y -22.1116,Z 65,A -37.7744,B 24.8617,C -2.7139,E1 25.1366,E2 121.1448} C_DIS
LIN {X 36.0349,Y -24.571,Z 65,A -41.789,B 24.8631,C -2.7001,E1 25.1304,E2 125.172} C_DIS
LIN {X 34.5277,Y -26.6471,Z 65,A -44.6768,B 24.8631,C -2.6995,E1 25.1256,E2 128.0473} C_DIS
LIN {X 33.1046,Y -28.396,Z 65,A -47.814,B 24.8642,C -2.6889,E1 25.12,E2 131.1952} C_DIS
LIN {X 31.418,Y -30.2512,Z 65,A -51.0801,B 24.865,C -2.6813,E1 25.1137,E2 134.465} C_DIS
LIN {X 29.6257,Y -32.0091,Z 65,A -54.4016,B 24.8658,C -2.6732,E1 25.107,E2 137.7919} C_DIS
LIN {X 27.75,Y -33.648,Z 65,A -57.6432,B 24.8665,C -2.6666,E1 25.1001,E2 141.0369} C_DIS
LIN {X 26.0105,Y -35.0104,Z 65,A -60.3326,B 24.8667,C -2.6641,E1 25.0941,E2 143.7223} C_DIS
LIN {X 23.9054,Y -36.4798,Z 65,A -64.0946,B 24.868,C -2.651,E1 25.0854,E2 147.5025} C_DIS
LIN {X 21.5164,Y -37.938,Z 65,A -67.6206,B 24.8684,C -2.6469,E1 25.0769,E2 151.0275} C_DIS
LIN {X 18.8983,Y -39.3075,Z 65,A -71.3308,B 24.8688,C -2.6435,E1 25.0677,E2 154.7358} C_DIS
LIN {X 17.0401,Y -40.1482,Z 65,A -74.2094,B 24.8695,C -2.6363,E1 25.0603,E2 157.6244} C_DIS
LIN {X 14.3861,Y -41.1736,Z 65,A -77.5914,B 24.8695,C -2.6371,E1 25.0514,E2 160.9973} C_DIS
LIN {X 12.6146,Y -41.7502,Z 65,A -80.225,B 24.87,C -2.6314,E1 25.0444,E2 163.6398} C_DIS
LIN {X 10.3372,Y -42.3718,Z 65,A -83.666,B 24.8708,C -2.6229,E1 25.0351,E2 167.0956} C_DIS
LIN {X 6.6095,Y -43.1108,Z 65,A -88.3352,B 24.8708,C -2.624,E1 25.0222,E2 171.757} C_DIS
LIN {X 4.1084,Y -43.4207,Z 65,A -91.591,B 24.8708,C -2.623,E1 25.0132,E2 175.0131} C_DIS
LIN {X 1.636,Y -43.5841,Z 65,A -94.5981,B 24.8706,C -2.6254,E1 25.0048,E2 178.0132} C_DIS
LIN {X 0.2144,Y -43.6138,Z 65,A -95.5654,B 24.8693,C -2.6386,E1 25.0022,E2 178.9492} C_DIS
Enddeposition()
LIN {X 0.2144,Y -43.6138,Z 65,A -95.5654,B 24.8693,C -2.6386,E1 25.0022,E2 178.9492} C_DIS
Startdeposition()
$VEL.CP = VEL_PRINT
LIN {X 1.3527,Y -42.6506,Z 65,A -93.8837,B 24.8674,C -2.6575,E1 25.0071,E2 177.2228} C_DIS
LIN {X 3.1218,Y -42.5581,Z 65,A -91.2629,B 24.8669,C -2.6622,E1 25.0144,E2 174.592} C_DIS
LIN {X 5.7599,Y -42.282,Z 65,A -88.0461,B 24.8672,C -2.659,E1 25.0233,E2 171.3851} C_DIS
LIN {X 8.4083,Y -41.8356,Z 65,A -83.7684,B 24.8659,C -2.6723,E1 25.0351,E2 167.0805} C_DIS
LIN {X 10.9582,Y -41.2414,Z 65,A -80.8358,B 24.8665,C -2.6666,E1 25.043,E2 164.166} C_DIS
LIN {X 12.9731,Y -40.6525,Z 65,A -77.7611,B 24.8657,C -2.6739,E1 25.0512,E2 161.0794} C_DIS
LIN {X 15.2095,Y -39.8695,Z 65,A -74.1086,B 24.8645,C -2.6857,E1 25.0608,E2 157.4067} C_DIS
LIN {X 17.6134,Y -38.8674,Z 65,A -71.1658,B 24.8649,C -2.6818,E1 25.0683,E2 154.4803} C_DIS
LIN {X 19.7709,Y -37.8157,Z 65,A -67.3576,B 24.8634,C -2.6967,E1 25.0778,E2 150.6473} C_DIS
LIN {X 22.1273,Y -36.4868,Z 65,A -64.4176,B 24.8639,C -2.6917,E1 25.0849,E2 147.7282} C_DIS
LIN {X 24.2648,Y -35.1017,Z 65,A -60.7321,B 24.8628,C -2.7027,E1 25.0934,E2 144.0288} C_DIS
LIN {X 26.0877,Y -33.7689,Z 65,A -58.0301,B 24.8628,C -2.7034,E1 25.0994,E2 141.3349} C_DIS
LIN {X 28.5212,Y -31.7396,Z 65,A -53.2834,B 24.8609,C -2.7213,E1 25.1095,E2 136.5645} C_DIS
LIN {X 31.1602,Y -29.154,Z 65,A -48.1522,B 24.8594,C -2.7361,E1 25.1195,E2 131.4201} C_DIS
LIN {X 33.2579,Y -26.7365,Z 65,A -44.7403,B 24.8599,C -2.7317,E1 25.1256,E2 128.0344} C_DIS
LIN {X 34.704,Y -24.8302,Z 65,A -41.0128,B 24.858,C -2.7492,E1 25.1318,E2 124.2833} C_DIS
LIN {X 36.2861,Y -22.4556,Z 65,A -36.9744,B 24.8566,C -2.7635,E1 25.1379,E2 120.2315} C_DIS
LIN {X 38.33,Y -18.7554,Z 65,A -31.7855,B 24.8558,C -2.7712,E1 25.1446,E2 115.0518} C_DIS
LIN {X 39.3628,Y -16.4767,Z 65,A -28.2556,B 24.8544,C -2.7842,E1 25.1486,E2 111.5104} C_DIS
LIN {X 40.3528,Y -13.8782,Z 65,A -24.7742,B 24.8537,C -2.791,E1 25.1519,E2 108.0324} C_DIS
LIN {X 40.9869,Y -11.8751,Z 65,A -22.1698,B 24.8532,C -2.7958,E1 25.154,E2 105.4315} C_DIS
LIN {X 41.6702,Y -9.1914,Z 65,A -17.6437,B 24.8504,C -2.8218,E1 25.1569,E2 100.87} C_DIS
LIN {X 42.327,Y -5.416,Z 65,A -13.2072,B 24.8501,C -2.8252,E1 25.1588,E2 96.4517} C_DIS
LIN {X 42.5577,Y -3.1324,Z 65,A -9.8919,B 24.8486,C -2.839,E1 25.1595,E2 93.1232} C_DIS
LIN {X 42.6668,Y -0.6768,Z 65,A -6.8718,B 24.848,C -2.8444,E1 25.1598,E2 90.1084} C_DIS
LIN {X 42.6355,Y 1.7674,Z 65,A -3.8446,B 24.8474,C -2.8501,E1 25.1596,E2 87.0856} C_DIS
LIN {X 42.5265,Y 3.5198,Z 65,A -1.4974,B 24.8466,C -2.8573,E1 25.1591,E2 84.7353} C_DIS
LIN {X 42.3566,Y 5.1827,Z 65,A 1.2606,B 24.8449,C -2.8734,E1 25.1582,E2 81.9556} C_DIS
LIN {X 41.9905,Y 7.5959,Z 65,A 4.8093,B 24.8433,C -2.8883,E1 25.1565,E2 78.3925} C_DIS
LIN {X 41.3542,Y 10.5235,Z 65,A 7.9891,B 24.8436,C -2.8854,E1 25.1545,E2 75.238} C_DIS
LIN {X 40.9346,Y 12.0527,Z 65,A 10.3306,B 24.8425,C -2.8954,E1 25.1527,E2 72.8861} C_DIS
LIN {X 40.2154,Y 14.2704,Z 65,A 13.2442,B 24.8419,C -2.9007,E1 25.15,E2 69.9764} C_DIS
LIN {X 39.6318,Y 15.8192,Z 65,A 15.9489,B 24.8403,C -2.9155,E1 25.1473,E2 67.2518} C_DIS
LIN {X 38.19,Y 19.0377,Z 65,A 19.9659,B 24.8403,C -2.916,E1 25.1426,E2 63.2552} C_DIS
LIN {X 37.0396,Y 21.189,Z 65,A 23.8839,B 24.838,C -2.9358,E1 25.1372,E2 59.3108} C_DIS
LIN {X 35.6945,Y 23.3841,Z 65,A 26.9851,B 24.8377,C -2.9385,E1 25.1326,E2 56.2189} C_DIS
LIN {X 34.6467,Y 24.9104,Z 65,A 29.3099,B 24.8374,C -2.9418,E1 25.1289,E2 53.8976} C_DIS
LIN {X 33.3656,Y 26.6018,Z 65,A 32.8672,B 24.8353,C -2.9605,E1 25.1227,E2 50.3126} C_DIS
LIN {X 31.6383,Y 28.6351,Z 65,A 35.9242,B 24.8353,C -2.9596,E1 25.1171,E2 47.2716} C_DIS
LIN {X 30.3009,Y 30.0461,Z 65,A 38.4685,B 24.8349,C -2.964,E1 25.1121,E2 44.7278} C_DIS
LIN {X 28.6071,Y 31.6634,Z 65,A 41.6939,B 24.834,C -2.9716,E1 25.1055,E2 41.4975} C_DIS
LIN {X 26.6529,Y 33.3255,Z 65,A 45.6593,B 24.8324,C -2.9865,E1 25.0969,E2 37.5118} C_DIS
LIN {X 23.7134,Y 35.4773,Z 65,A 49.6874,B 24.833,C -2.9804,E1 25.0878,E2 33.512} C_DIS
LIN {X 22.5291,Y 36.2402,Z 65,A 51.8512,B 24.8322,C -2.9877,E1 25.0826,E2 31.338} C_DIS
LIN {X 20.5437,Y 37.402,Z 65,A 55.0819,B 24.8315,C -2.9942,E1 25.0748,E2 28.1014} C_DIS
LIN {X 17.8404,Y 38.7641,Z 65,A 58.5554,B 24.832,C -2.9897,E1 25.0661,E2 24.6477} C_DIS
LIN {X 16.2222,Y 39.4685,Z 65,A 61.5463,B 24.8306,C -3.0019,E1 25.0584,E2 21.6349} C_DIS
LIN {X 13.4425,Y 40.4999,Z 65,A 65.1123,B 24.831,C -2.9989,E1 25.049,E2 18.0832} C_DIS
LIN {X 11.0466,Y 41.2175,Z 65,A 68.9599,B 24.8299,C -3.0086,E1 25.0386,E2 14.2191} C_DIS
LIN {X 8.5187,Y 41.8131,Z 65,A 71.7219,B 24.8309,C -2.9994,E1 25.0312,E2 11.4825} C_DIS
LIN {X 6.4101,Y 42.1878,Z 65,A 75.1126,B 24.8299,C -3.008,E1 25.0218,E2 8.0749} C_DIS
LIN {X 4.2686,Y 42.4582,Z 65,A 77.6392,B 24.8305,C -3.003,E1 25.0148,E2 5.562} C_DIS
LIN {X 1.9666,Y 42.6269,Z 65,A 81.3555,B 24.8295,C -3.0119,E1 25.0044,E2 1.8259} C_DIS
LIN {X -0.474,Y 42.6699,Z 65,A 84.1876,B 24.8303,C -3.0049,E1 24.9965,E2 -0.9893} C_DIS
LIN {X -2.7891,Y 42.5809,Z 65,A 87.4362,B 24.8302,C -3.0057,E1 24.9875,E2 -4.2408} C_DIS
LIN {X -5.1437,Y 42.3613,Z 65,A 90.6544,B 24.8303,C -3.0046,E1 24.9785,E2 -7.4584} C_DIS
LIN {X -7.6158,Y 41.987,Z 65,A 93.8106,B 24.8309,C -2.9995,E1 24.9699,E2 -10.6054} C_DIS
LIN {X -9.4167,Y 41.6205,Z 65,A 96.3776,B 24.8309,C -2.9988,E1 24.9629,E2 -13.1737} C_DIS
LIN {X -11.5833,Y 41.0698,Z 65,A 99.4721,B 24.8312,C -2.997,E1 24.9545,E2 -16.2687} C_DIS
LIN {X -13.2379,Y 40.5669,Z 65,A 101.6404,B 24.8317,C -2.9923,E1 24.9488,E2 -18.4297} C_DIS
LIN {X -15.5088,Y 39.7541,Z 65,A 105.1177,B 24.8318,C -2.9914,E1 24.9397,E2 -21.9119} C_DIS
LIN {X -17.4467,Y 38.9425,Z 65,A 107.5596,B 24.8328,C -2.9824,E1 24.9334,E2 -24.3381} C_DIS
LIN {X -19.3287,Y 38.0436,Z 65,A 110.8701,B 24.8326,C -2.9846,E1 24.9251,E2 -27.6626} C_DIS
LIN {X -21.3987,Y 36.9191,Z 65,A 114.069,B 24.8331,C -2.9796,E1 24.9174,E2 -30.859} C_DIS
LIN {X -23.4346,Y 35.6612,Z 65,A 117.1926,B 24.8339,C -2.9725,E1 24.91,E2 -33.9758} C_DIS
LIN {X -25.9973,Y 33.8385,Z 65,A 121.3541,B 24.835,C -2.9633,E1 24.9007,E2 -38.1299} C_DIS
LIN {X -27.9209,Y 32.2702,Z 65,A 124.73,B 24.8357,C -2.9566,E1 24.8935,E2 -41.5028} C_DIS
LIN {X -29.904,Y 30.4412,Z 65,A 128.2088,B 24.8368,C -2.9465,E1 24.8865,E2 -44.9718} C_DIS
LIN {X -31.2836,Y 29.0223,Z 65,A 131.0583,B 24.8373,C -2.9424,E1 24.881,E2 -47.8239} C_DIS
LIN {X -33.1506,Y 26.869,Z 65,A 134.5645,B 24.8388,C -2.929,E1 24.8747,E2 -51.314} C_DIS
LIN {X -34.47,Y 25.1541,Z 65,A 137.7533,B 24.8393,C -2.9247,E1 24.8693,E2 -54.5078} C_DIS
LIN {X -35.8718,Y 23.111,Z 65,A 141.1338,B 24.8402,C -2.9163,E1 24.8641,E2 -57.8851} C_DIS
LIN {X -37.0942,Y 21.0933,Z 65,A 144.0655,B 24.8415,C -2.9047,E1 24.86,E2 -60.8042} C_DIS
LIN {X -38.0444,Y 19.327,Z 65,A 146.9526,B 24.8421,C -2.8992,E1 24.8563,E2 -63.6936} C_DIS
LIN {X -39.3935,Y 16.4023,Z 65,A 151.1202,B 24.8437,C -2.8846,E1 24.8515,E2 -67.8493} C_DIS
LIN {X -40.0117,Y 14.8328,Z 65,A 153.7159,B 24.844,C -2.8816,E1 24.8489,E2 -70.4524} C_DIS
LIN {X -40.906,Y 12.1491,Z 65,A 157.4144,B 24.8454,C -2.8689,E1 24.8458,E2 -74.1417} C_DIS
LIN {X -41.6191,Y 9.4173,Z 65,A 161.1096,B 24.8467,C -2.8561,E1 24.8434,E2 -77.8278} C_DIS
LIN {X -42.0702,Y 7.1399,Z 65,A 164.6315,B 24.8473,C -2.851,E1 24.8416,E2 -81.3584} C_DIS
LIN {X -42.5761,Y 2.8596,Z 65,A 171.1241,B 24.8484,C -2.8409,E1 24.8399,E2 -87.8659} C_DIS
LIN {X -42.6578,Y -1.1187,Z 65,A 176.0733,B 24.8506,C -2.8196,E1 24.8399,E2 -92.7938} C_DIS
LIN {X -42.4113,Y -4.7167,Z 65,A -178.8091,B 24.8519,C -2.8078,E1 24.8413,E2 -97.9138} C_DIS
LIN {X -41.7386,Y -8.8794,Z 65,A -174.1066,B 24.8549,C -2.7794,E1 24.8436,E2 -102.5763} C_DIS
LIN {X -41.125,Y -11.3868,Z 65,A -170.0612,B 24.8553,C -2.7758,E1 24.8464,E2 -106.6366} C_DIS
LIN {X -40.3622,Y -13.8494,Z 65,A -166.6876,B 24.8564,C -2.7647,E1 24.8494,E2 -110.0029} C_DIS
LIN {X -39.3132,Y -16.5944,Z 65,A -163.0219,B 24.8579,C -2.7502,E1 24.8531,E2 -113.6546} C_DIS
LIN {X -38.4432,Y -18.5209,Z 65,A -159.4992,B 24.8579,C -2.7506,E1 24.8574,E2 -117.1972} C_DIS
LIN {X -36.9328,Y -21.3745,Z 65,A -155.267,B 24.8592,C -2.7379,E1 24.8631,E2 -121.4214} C_DIS
LIN {X -35.5944,Y -23.5359,Z 65,A -152.3728,B 24.8607,C -2.723,E1 24.8674,E2 -124.2946} C_DIS
LIN {X -34.3901,Y -25.2631,Z 65,A -149.3766,B 24.8612,C -2.7182,E1 24.8723,E2 -127.294} C_DIS
LIN {X -32.9528,Y -27.1115,Z 65,A -145.3688,B 24.8609,C -2.7217,E1 24.8794,E2 -131.3288} C_DIS
LIN {X -30.4931,Y -29.8515,Z 65,A -141.1174,B 24.8628,C -2.7024,E1 24.8875,E2 -135.5527} C_DIS
LIN {X -28.485,Y -31.7728,Z 65,A -137.5081,B 24.8638,C -2.6935,E1 24.8949,E2 -139.1554} C_DIS
LIN {X -26.8621,Y -33.1561,Z 65,A -134.6773,B 24.8643,C -2.6879,E1 24.9009,E2 -141.9835} C_DIS
LIN {X -25.3488,Y -34.3273,Z 65,A -131.8539,B 24.8644,C -2.6868,E1 24.9073,E2 -144.8144} C_DIS
LIN {X -23.0476,Y -35.9125,Z 65,A -128.5745,B 24.8657,C -2.6747,E1 24.9148,E2 -148.076} C_DIS
LIN {X -21.7305,Y -36.7245,Z 65,A -125.8095,B 24.865,C -2.6809,E1 24.9215,E2 -150.8641} C_DIS
LIN {X -19.3518,Y -38.0318,Z 65,A -122.4309,B 24.8659,C -2.6727,E1 24.9298,E2 -154.2325} C_DIS
LIN {X -16.3554,Y -39.4139,Z 65,A -118.3112,B 24.8668,C -2.6637,E1 24.9403,E2 -158.3407} C_DIS
LIN {X -14.1195,Y -40.2684,Z 65,A -114.5772,B 24.8663,C -2.6682,E1 24.9501,E2 -162.0928} C_DIS
LIN {X -12.1321,Y -40.911,Z 65,A -112.0042,B 24.8668,C -2.6629,E1 24.957,E2 -164.6579} C_DIS
LIN {X -8.7534,Y -41.765,Z 65,A -107.1554,B 24.8668,C -2.663,E1 24.9702,E2 -169.5133} C_DIS
LIN {X -6.3755,Y -42.1933,Z 65,A -104.1591,B 24.8673,C -2.6585,E1 24.9784,E2 -172.5017} C_DIS
LIN {X -4.0965,Y -42.4753,Z 65,A -101.3036,B 24.8677,C -2.6548,E1 24.9863,E2 -175.3501} C_DIS
LIN {X -2.699,Y -42.587,Z 65,A -99.2263,B 24.8674,C -2.6577,E1 24.9921,E2 -177.4351} C_DIS
LIN {X -0.6654,Y -42.6665,Z 65,A -96.544,B 24.8674,C -2.6573,E1 24.9996,E2 -180.1169} C_DIS
LIN {X -0.6654,Y -42.6665,Z 65,A -96.544,B 24.8674,C -2.6573,E1 24.9996,E2 -180.1169} C_DIS
Enddeposition()
LIN {X 0.2084,Y -41.7255,Z 65,A -95.7173,B 24.8663,C -2.6687,E1 25.002,E2 -180.9706} C_DIS
Startdeposition()
$VEL.CP = VEL_PRINT
LIN {X -1.5179,Y -41.7015,Z 65,A -99.012,B 24.8676,C -2.655,E1 24.9927,E2 -177.643} C_DIS
LIN {X -3.215,Y -41.6057,Z 65,A -101.8929,B 24.8684,C -2.6473,E1 24.9846,E2 -174.7428} C_DIS
LIN {X -6.5978,Y -41.2053,Z 65,A -106.1891,B 24.8678,C -2.6535,E1 24.9728,E2 -170.4579} C_DIS
LIN {X -8.9799,Y -40.752,Z 65,A -109.6039,B 24.8678,C -2.6537,E1 24.9634,E2 -167.0397} C_DIS
LIN {X -11.1678,Y -40.208,Z 65,A -112.3549,B 24.8671,C -2.6601,E1 24.956,E2 -164.2998} C_DIS
LIN {X -13.2884,Y -39.5572,Z 65,A -115.8704,B 24.8675,C -2.6562,E1 24.9466,E2 -160.7686} C_DIS
LIN {X -15.3332,Y -38.8105,Z 65,A -118.2773,B 24.8665,C -2.6665,E1 24.9404,E2 -158.3812} C_DIS
LIN {X -16.7441,Y -38.223,Z 65,A -120.6952,B 24.8667,C -2.6645,E1 24.9342,E2 -155.9529} C_DIS
LIN {X -18.8171,Y -37.2466,Z 65,A -123.8855,B 24.8664,C -2.6676,E1 24.9262,E2 -152.7618} C_DIS
LIN {X -21.1622,Y -35.9656,Z 65,A -127.5634,B 24.8659,C -2.6724,E1 24.9172,E2 -149.0847} C_DIS
LIN {X -22.9664,Y -34.841,Z 65,A -130.4797,B 24.8654,C -2.6768,E1 24.9104,E2 -146.1696} C_DIS
LIN {X -25.1462,Y -33.3022,Z 65,A -134.0715,B 24.8647,C -2.6838,E1 24.9023,E2 -142.5818} C_DIS
LIN {X -27.5338,Y -31.3569,Z 65,A -138.1804,B 24.8638,C -2.693,E1 24.8935,E2 -138.4791} C_DIS
LIN {X -28.8415,Y -30.1587,Z 65,A -140.9511,B 24.8638,C -2.6938,E1 24.8878,E2 -135.699} C_DIS
LIN {X -30.5762,Y -28.3992,Z 65,A -144.7652,B 24.8635,C -2.696,E1 24.8804,E2 -131.8738} C_DIS
LIN {X -32.4251,Y -26.2672,Z 65,A -148.0653,B 24.8619,C -2.7115,E1 24.8745,E2 -128.5954} C_DIS
LIN {X -33.833,Y -24.4271,Z 65,A -151.6615,B 24.8616,C -2.7143,E1 24.8685,E2 -124.9886} C_DIS
LIN {X -35.1097,Y -22.5536,Z 65,A -154.8924,B 24.861,C -2.7208,E1 24.8636,E2 -121.7569} C_DIS
LIN {X -36.6613,Y -19.9325,Z 65,A -158.7903,B 24.8595,C -2.7349,E1 24.8582,E2 -117.8724} C_DIS
LIN {X -37.6256,Y -18.0464,Z 65,A -161.7015,B 24.8587,C -2.7428,E1 24.8546,E2 -114.9643} C_DIS
LIN {X -38.5891,Y -15.8827,Z 65,A -165.4811,B 24.8584,C -2.7461,E1 24.8505,E2 -111.1717} C_DIS
LIN {X -39.6091,Y -13.1346,Z 65,A -168.9153,B 24.8565,C -2.7641,E1 24.8474,E2 -107.7612} C_DIS
LIN {X -40.2131,Y -11.1497,Z 65,A -171.4352,B 24.8552,C -2.7761,E1 24.8454,E2 -105.2554} C_DIS
LIN {X -40.6377,Y -9.4836,Z 65,A -174.2997,B 24.8551,C -2.7777,E1 24.8435,E2 -102.3779} C_DIS
LIN {X -41.2084,Y -6.5723,Z 65,A -178.3373,B 24.8537,C -2.7905,E1 24.8415,E2 -98.347} C_DIS
LIN {X -41.476,Y -4.5947,Z 65,A 179.0382,B 24.8527,C -2.8002,E1 24.8406,E2 -95.7301} C_DIS
LIN {X -41.6543,Y -2.5144,Z 65,A 175.9362,B 24.852,C -2.8066,E1 24.8399,E2 -92.6246} C_DIS
LIN {X -41.7297,Y -0.0668,Z 65,A 172.6437,B 24.8508,C -2.8178,E1 24.8398,E2 -89.3393} C_DIS
LIN {X -41.6188,Y 3.0477,Z 65,A 167.9085,B 24.8499,C -2.8264,E1 24.8405,E2 -84.5962} C_DIS
LIN {X -41.3479,Y 5.636,Z 65,A 164.0624,B 24.849,C -2.8347,E1 24.8418,E2 -80.7469} C_DIS
LIN {X -40.6569,Y 9.4005,Z 65,A 159.9712,B 24.8459,C -2.8635,E1 24.844,E2 -76.7005} C_DIS
LIN {X -40.2737,Y 10.9265,Z 65,A 157.2407,B 24.8459,C -2.864,E1 24.846,E2 -73.9554} C_DIS
LIN {X -39.5894,Y 13.1929,Z 65,A 153.8559,B 24.845,C -2.8725,E1 24.8488,E2 -70.5713} C_DIS
LIN {X -38.7236,Y 15.5523,Z 65,A 150.4761,B 24.8438,C -2.8836,E1 24.8522,E2 -67.1991} C_DIS
LIN {X -37.7292,Y 17.8304,Z 65,A 147.0093,B 24.8427,C -2.893,E1 24.8562,E2 -63.7358} C_DIS
LIN {X -36.4443,Y 20.3266,Z 65,A 142.5574,B 24.8422,C -2.8976,E1 24.8621,E2 -59.2713} C_DIS
LIN {X -35.1697,Y 22.4601,Z 65,A 139.6515,B 24.8406,C -2.9125,E1 24.8664,E2 -56.3863} C_DIS
LIN {X -33.7927,Y 24.4837,Z 65,A 136.3634,B 24.8395,C -2.9223,E1 24.8716,E2 -53.1055} C_DIS
Enddeposition()
END
